LIN {X 226.458,Y -181.154,Z 168.975,A 141.342,B 90.000,C 0.000} C_DIS
LIN {X 226.330,Y -181.313,Z 169.018,A 141.302,B 90.000,C 0.000} C_DIS
LIN {X 226.304,Y -181.347,Z 169.069,A 141.293,B 90.000,C 0.000} C_DIS
LIN {X 226.264,Y -181.396,Z 169.120,A 141.281,B 90.000,C 0.000} C_DIS
LIN {X 226.072,Y -181.635,Z 169.162,A 141.220,B 90.000,C 0.000} C_DIS
LIN {X 225.993,Y -181.734,Z 169.264,A 141.195,B 90.000,C 0.000} C_DIS
LIN {X 225.801,Y -181.973,Z 169.307,A 141.135,B 90.000,C 0.000} C_DIS
LIN {X 225.721,Y -182.072,Z 169.409,A 141.109,B 90.000,C 0.000} C_DIS
LIN {X 225.528,Y -182.310,Z 169.451,A 141.049,B 90.000,C 0.000} C_DIS
LIN {X 225.488,Y -182.360,Z 169.502,A 141.036,B 90.000,C 0.000} C_DIS
LIN {X 225.461,Y -182.393,Z 169.554,A 141.028,B 90.000,C 0.000} C_DIS
LIN {X 225.333,Y -182.551,Z 169.596,A 140.988,B 90.000,C 0.000} C_DIS
LIN {X 225.306,Y -182.584,Z 169.647,A 140.979,B 90.000,C 0.000} C_DIS
LIN {X 225.266,Y -182.634,Z 169.698,A 140.967,B 90.000,C 0.000} C_DIS
LIN {X 225.073,Y -182.872,Z 169.740,A 140.906,B 90.000,C 0.000} C_DIS
LIN {X 224.993,Y -182.970,Z 169.843,A 140.881,B 90.000,C 0.000} C_DIS
LIN {X 224.800,Y -183.208,Z 169.885,A 140.821,B 90.000,C 0.000} C_DIS
LIN {X 224.719,Y -183.307,Z 169.987,A 140.795,B 90.000,C 0.000} C_DIS
LIN {X 224.525,Y -183.544,Z 170.030,A 140.735,B 90.000,C 0.000} C_DIS
LIN {X 224.445,Y -183.642,Z 170.132,A 140.710,B 90.000,C 0.000} C_DIS
LIN {X 224.251,Y -183.879,Z 170.174,A 140.649,B 90.000,C 0.000} C_DIS
LIN {X 224.210,Y -183.929,Z 170.225,A 140.637,B 90.000,C 0.000} C_DIS
LIN {X 224.183,Y -183.961,Z 170.276,A 140.628,B 90.000,C 0.000} C_DIS
LIN {X 224.054,Y -184.119,Z 170.319,A 140.588,B 90.000,C 0.000} C_DIS
LIN {X 224.027,Y -184.152,Z 170.370,A 140.580,B 90.000,C 0.000} C_DIS
LIN {X 223.986,Y -184.201,Z 170.421,A 140.567,B 90.000,C 0.000} C_DIS
LIN {X 223.792,Y -184.438,Z 170.463,A 140.506,B 90.000,C 0.000} C_DIS
LIN {X 223.711,Y -184.536,Z 170.565,A 140.481,B 90.000,C 0.000} C_DIS
LIN {X 223.516,Y -184.772,Z 170.608,A 140.421,B 90.000,C 0.000} C_DIS
LIN {X 223.435,Y -184.870,Z 170.710,A 140.396,B 90.000,C 0.000} C_DIS
LIN {X 223.239,Y -185.106,Z 170.752,A 140.335,B 90.000,C 0.000} C_DIS
LIN {X 223.199,Y -185.155,Z 170.803,A 140.323,B 90.000,C 0.000} C_DIS
LIN {X 223.172,Y -185.188,Z 170.854,A 140.314,B 90.000,C 0.000} C_DIS
LIN {X 223.041,Y -185.345,Z 170.897,A 140.274,B 90.000,C 0.000} C_DIS
LIN {X 223.014,Y -185.377,Z 170.948,A 140.265,B 90.000,C 0.000} C_DIS
LIN {X 222.973,Y -185.426,Z 170.999,A 140.253,B 90.000,C 0.000} C_DIS
LIN {X 222.777,Y -185.662,Z 171.041,A 140.192,B 90.000,C 0.000} C_DIS
LIN {X 222.696,Y -185.759,Z 171.143,A 140.167,B 90.000,C 0.000} C_DIS
LIN {X 222.500,Y -185.995,Z 171.186,A 140.107,B 90.000,C 0.000} C_DIS
LIN {X 222.418,Y -186.092,Z 171.288,A 140.082,B 90.000,C 0.000} C_DIS
LIN {X 222.221,Y -186.327,Z 171.330,A 140.021,B 90.000,C 0.000} C_DIS
LIN {X 222.180,Y -186.376,Z 171.381,A 140.008,B 90.000,C 0.000} C_DIS
LIN {X 222.153,Y -186.408,Z 171.432,A 140.000,B 90.000,C 0.000} C_DIS
LIN {X 222.022,Y -186.565,Z 171.475,A 139.960,B 90.000,C 0.000} C_DIS
LIN {X 221.994,Y -186.597,Z 171.526,A 139.951,B 90.000,C 0.000} C_DIS
LIN {X 221.953,Y -186.646,Z 171.577,A 139.939,B 90.000,C 0.000} C_DIS
LIN {X 221.756,Y -186.880,Z 171.619,A 139.878,B 90.000,C 0.000} C_DIS
LIN {X 221.674,Y -186.977,Z 171.721,A 139.853,B 90.000,C 0.000} C_DIS
LIN {X 221.477,Y -187.211,Z 171.764,A 139.793,B 90.000,C 0.000} C_DIS
LIN {X 221.394,Y -187.309,Z 171.866,A 139.767,B 90.000,C 0.000} C_DIS
LIN {X 221.196,Y -187.542,Z 171.908,A 139.707,B 90.000,C 0.000} C_DIS
LIN {X 221.114,Y -187.640,Z 172.010,A 139.682,B 90.000,C 0.000} C_DIS
LIN {X 220.916,Y -187.873,Z 172.053,A 139.621,B 90.000,C 0.000} C_DIS
LIN {X 220.875,Y -187.921,Z 172.104,A 139.609,B 90.000,C 0.000} C_DIS
LIN {X 220.847,Y -187.954,Z 172.155,A 139.600,B 90.000,C 0.000} C_DIS
LIN {X 220.715,Y -188.109,Z 172.197,A 139.560,B 90.000,C 0.000} C_DIS
LIN {X 220.687,Y -188.141,Z 172.249,A 139.552,B 90.000,C 0.000} C_DIS
LIN {X 220.646,Y -188.190,Z 172.300,A 139.539,B 90.000,C 0.000} C_DIS
LIN {X 220.447,Y -188.423,Z 172.342,A 139.478,B 90.000,C 0.000} C_DIS
LIN {X 220.364,Y -188.520,Z 172.444,A 139.453,B 90.000,C 0.000} C_DIS
LIN {X 220.165,Y -188.752,Z 172.487,A 139.393,B 90.000,C 0.000} C_DIS
LIN {X 220.082,Y -188.849,Z 172.589,A 139.368,B 90.000,C 0.000} C_DIS
LIN {X 219.883,Y -189.081,Z 172.631,A 139.307,B 90.000,C 0.000} C_DIS
LIN {X 219.841,Y -189.129,Z 172.682,A 139.295,B 90.000,C 0.000} C_DIS
LIN {X 219.813,Y -189.162,Z 172.733,A 139.286,B 90.000,C 0.000} C_DIS
LIN {X 219.680,Y -189.316,Z 172.776,A 139.246,B 90.000,C 0.000} C_DIS
LIN {X 219.652,Y -189.348,Z 172.827,A 139.237,B 90.000,C 0.000} C_DIS
LIN {X 219.611,Y -189.397,Z 172.878,A 139.225,B 90.000,C 0.000} C_DIS
LIN {X 219.411,Y -189.628,Z 172.920,A 139.164,B 90.000,C 0.000} C_DIS
LIN {X 219.327,Y -189.725,Z 173.022,A 139.139,B 90.000,C 0.000} C_DIS
LIN {X 219.127,Y -189.956,Z 173.065,A 139.079,B 90.000,C 0.000} C_DIS
LIN {X 219.043,Y -190.053,Z 173.167,A 139.054,B 90.000,C 0.000} C_DIS
LIN {X 218.843,Y -190.284,Z 173.209,A 138.993,B 90.000,C 0.000} C_DIS
LIN {X 218.801,Y -190.332,Z 173.260,A 138.980,B 90.000,C 0.000} C_DIS
LIN {X 218.773,Y -190.364,Z 173.311,A 138.972,B 90.000,C 0.000} C_DIS
LIN {X 218.639,Y -190.518,Z 173.354,A 138.932,B 90.000,C 0.000} C_DIS
LIN {X 218.611,Y -190.550,Z 173.405,A 138.923,B 90.000,C 0.000} C_DIS
LIN {X 218.569,Y -190.598,Z 173.456,A 138.911,B 90.000,C 0.000} C_DIS
LIN {X 218.368,Y -190.828,Z 173.498,A 138.850,B 90.000,C 0.000} C_DIS
LIN {X 218.284,Y -190.924,Z 173.600,A 138.825,B 90.000,C 0.000} C_DIS
LIN {X 218.082,Y -191.155,Z 173.643,A 138.765,B 90.000,C 0.000} C_DIS
LIN {X 217.998,Y -191.250,Z 173.745,A 138.739,B 90.000,C 0.000} C_DIS
LIN {X 217.796,Y -191.481,Z 173.787,A 138.679,B 90.000,C 0.000} C_DIS
LIN {X 217.712,Y -191.576,Z 173.889,A 138.654,B 90.000,C 0.000} C_DIS
LIN {X 217.510,Y -191.806,Z 173.932,A 138.593,B 90.000,C 0.000} C_DIS
LIN {X 217.468,Y -191.854,Z 173.983,A 138.581,B 90.000,C 0.000} C_DIS
LIN {X 217.439,Y -191.886,Z 174.034,A 138.572,B 90.000,C 0.000} C_DIS
LIN {X 217.304,Y -192.039,Z 174.076,A 138.532,B 90.000,C 0.000} C_DIS
LIN {X 217.276,Y -192.070,Z 174.127,A 138.524,B 90.000,C 0.000} C_DIS
LIN {X 217.234,Y -192.118,Z 174.178,A 138.511,B 90.000,C 0.000} C_DIS
LIN {X 217.031,Y -192.347,Z 174.221,A 138.450,B 90.000,C 0.000} C_DIS
LIN {X 216.947,Y -192.443,Z 174.323,A 138.425,B 90.000,C 0.000} C_DIS
LIN {X 216.743,Y -192.672,Z 174.365,A 138.365,B 90.000,C 0.000} C_DIS
LIN {X 216.659,Y -192.767,Z 174.467,A 138.340,B 90.000,C 0.000} C_DIS
LIN {X 216.455,Y -192.996,Z 174.510,A 138.279,B 90.000,C 0.000} C_DIS
LIN {X 216.413,Y -193.043,Z 174.561,A 138.267,B 90.000,C 0.000} C_DIS
LIN {X 216.384,Y -193.075,Z 174.612,A 138.258,B 90.000,C 0.000} C_DIS
LIN {X 216.248,Y -193.227,Z 174.654,A 138.218,B 90.000,C 0.000} C_DIS
LIN {X 216.220,Y -193.259,Z 174.705,A 138.209,B 90.000,C 0.000} C_DIS
LIN {X 216.178,Y -193.306,Z 174.757,A 138.197,B 90.000,C 0.000} C_DIS
LIN {X 215.973,Y -193.534,Z 174.799,A 138.136,B 90.000,C 0.000} C_DIS
LIN {X 215.888,Y -193.629,Z 174.901,A 138.111,B 90.000,C 0.000} C_DIS
LIN {X 215.684,Y -193.857,Z 174.944,A 138.051,B 90.000,C 0.000} C_DIS
LIN {X 215.599,Y -193.952,Z 175.046,A 138.026,B 90.000,C 0.000} C_DIS
LIN {X 215.394,Y -194.179,Z 175.088,A 137.965,B 90.000,C 0.000} C_DIS
LIN {X 215.351,Y -194.227,Z 175.139,A 137.952,B 90.000,C 0.000} C_DIS
LIN {X 215.323,Y -194.258,Z 175.190,A 137.944,B 90.000,C 0.000} C_DIS
LIN {X 215.186,Y -194.410,Z 175.233,A 137.904,B 90.000,C 0.000} C_DIS
LIN {X 215.157,Y -194.441,Z 175.284,A 137.895,B 90.000,C 0.000} C_DIS
LIN {X 215.115,Y -194.488,Z 175.335,A 137.883,B 90.000,C 0.000} C_DIS
LIN {X 214.909,Y -194.715,Z 175.377,A 137.822,B 90.000,C 0.000} C_DIS
LIN {X 214.824,Y -194.810,Z 175.479,A 137.797,B 90.000,C 0.000} C_DIS
LIN {X 214.618,Y -195.036,Z 175.522,A 137.737,B 90.000,C 0.000} C_DIS
LIN {X 214.532,Y -195.131,Z 175.624,A 137.711,B 90.000,C 0.000} C_DIS
LIN {X 214.326,Y -195.357,Z 175.666,A 137.651,B 90.000,C 0.000} C_DIS
LIN {X 214.283,Y -195.404,Z 175.717,A 137.638,B 90.000,C 0.000} C_DIS
LIN {X 214.254,Y -195.436,Z 175.768,A 137.630,B 90.000,C 0.000} C_DIS
LIN {X 214.117,Y -195.586,Z 175.811,A 137.590,B 90.000,C 0.000} C_DIS
LIN {X 214.088,Y -195.618,Z 175.862,A 137.581,B 90.000,C 0.000} C_DIS
LIN {X 214.045,Y -195.665,Z 175.913,A 137.569,B 90.000,C 0.000} C_DIS
LIN {X 213.838,Y -195.891,Z 175.955,A 137.508,B 90.000,C 0.000} C_DIS
LIN {X 213.752,Y -195.984,Z 176.057,A 137.483,B 90.000,C 0.000} C_DIS
LIN {X 213.545,Y -196.210,Z 176.100,A 137.423,B 90.000,C 0.000} C_DIS
LIN {X 213.459,Y -196.304,Z 176.202,A 137.397,B 90.000,C 0.000} C_DIS
LIN {X 213.252,Y -196.529,Z 176.244,A 137.337,B 90.000,C 0.000} C_DIS
LIN {X 213.209,Y -196.576,Z 176.295,A 137.324,B 90.000,C 0.000} C_DIS
LIN {X 213.180,Y -196.607,Z 176.346,A 137.316,B 90.000,C 0.000} C_DIS
LIN {X 213.041,Y -196.757,Z 176.389,A 137.276,B 90.000,C 0.000} C_DIS
LIN {X 213.013,Y -196.788,Z 176.440,A 137.267,B 90.000,C 0.000} C_DIS
LIN {X 212.969,Y -196.835,Z 176.491,A 137.255,B 90.000,C 0.000} C_DIS
LIN {X 212.761,Y -197.060,Z 176.533,A 137.194,B 90.000,C 0.000} C_DIS
LIN {X 212.675,Y -197.153,Z 176.635,A 137.169,B 90.000,C 0.000} C_DIS
LIN {X 212.466,Y -197.378,Z 176.678,A 137.108,B 90.000,C 0.000} C_DIS
LIN {X 212.380,Y -197.471,Z 176.780,A 137.083,B 90.000,C 0.000} C_DIS
LIN {X 212.171,Y -197.695,Z 176.822,A 137.023,B 90.000,C 0.000} C_DIS
LIN {X 212.084,Y -197.788,Z 176.924,A 136.998,B 90.000,C 0.000} C_DIS
LIN {X 211.875,Y -198.012,Z 176.967,A 136.937,B 90.000,C 0.000} C_DIS
LIN {X 211.832,Y -198.059,Z 177.018,A 136.925,B 90.000,C 0.000} C_DIS
LIN {X 211.803,Y -198.090,Z 177.069,A 136.916,B 90.000,C 0.000} C_DIS
LIN {X 211.663,Y -198.239,Z 177.111,A 136.876,B 90.000,C 0.000} C_DIS
LIN {X 211.634,Y -198.270,Z 177.162,A 136.867,B 90.000,C 0.000} C_DIS
LIN {X 211.591,Y -198.316,Z 177.213,A 136.855,B 90.000,C 0.000} C_DIS
LIN {X 211.381,Y -198.540,Z 177.256,A 136.794,B 90.000,C 0.000} C_DIS
LIN {X 211.294,Y -198.632,Z 177.358,A 136.769,B 90.000,C 0.000} C_DIS
LIN {X 211.084,Y -198.855,Z 177.400,A 136.709,B 90.000,C 0.000} C_DIS
LIN {X 210.997,Y -198.948,Z 177.503,A 136.683,B 90.000,C 0.000} C_DIS
LIN {X 210.787,Y -199.171,Z 177.545,A 136.623,B 90.000,C 0.000} C_DIS
LIN {X 210.743,Y -199.217,Z 177.596,A 136.610,B 90.000,C 0.000} C_DIS
LIN {X 210.714,Y -199.248,Z 177.647,A 136.602,B 90.000,C 0.000} C_DIS
LIN {X 210.573,Y -199.396,Z 177.690,A 136.562,B 90.000,C 0.000} C_DIS
LIN {X 210.544,Y -199.427,Z 177.741,A 136.553,B 90.000,C 0.000} C_DIS
LIN {X 210.500,Y -199.473,Z 177.792,A 136.541,B 90.000,C 0.000} C_DIS
LIN {X 210.290,Y -199.695,Z 177.834,A 136.480,B 90.000,C 0.000} C_DIS
LIN {X 210.202,Y -199.788,Z 177.936,A 136.455,B 90.000,C 0.000} C_DIS
LIN {X 209.991,Y -200.010,Z 177.979,A 136.395,B 90.000,C 0.000} C_DIS
LIN {X 209.903,Y -200.102,Z 178.081,A 136.369,B 90.000,C 0.000} C_DIS
LIN {X 209.692,Y -200.323,Z 178.123,A 136.309,B 90.000,C 0.000} C_DIS
LIN {X 209.604,Y -200.415,Z 178.225,A 136.284,B 90.000,C 0.000} C_DIS
LIN {X 209.392,Y -200.637,Z 178.268,A 136.223,B 90.000,C 0.000} C_DIS
LIN {X 209.348,Y -200.683,Z 178.319,A 136.211,B 90.000,C 0.000} C_DIS
LIN {X 209.318,Y -200.713,Z 178.370,A 136.202,B 90.000,C 0.000} C_DIS
LIN {X 209.177,Y -200.861,Z 178.412,A 136.162,B 90.000,C 0.000} C_DIS
LIN {X 209.148,Y -200.891,Z 178.463,A 136.154,B 90.000,C 0.000} C_DIS
LIN {X 209.104,Y -200.937,Z 178.514,A 136.141,B 90.000,C 0.000} C_DIS
LIN {X 208.891,Y -201.158,Z 178.557,A 136.080,B 90.000,C 0.000} C_DIS
LIN {X 208.803,Y -201.250,Z 178.659,A 136.055,B 90.000,C 0.000} C_DIS
LIN {X 208.590,Y -201.470,Z 178.701,A 135.995,B 90.000,C 0.000} C_DIS
LIN {X 208.502,Y -201.561,Z 178.803,A 135.970,B 90.000,C 0.000} C_DIS
LIN {X 208.289,Y -201.782,Z 178.846,A 135.909,B 90.000,C 0.000} C_DIS
LIN {X 208.244,Y -201.827,Z 178.897,A 135.897,B 90.000,C 0.000} C_DIS
LIN {X 208.215,Y -201.858,Z 178.948,A 135.888,B 90.000,C 0.000} C_DIS
LIN {X 208.073,Y -202.004,Z 178.990,A 135.848,B 90.000,C 0.000} C_DIS
LIN {X 208.043,Y -202.035,Z 179.041,A 135.839,B 90.000,C 0.000} C_DIS
LIN {X 207.999,Y -202.080,Z 179.092,A 135.827,B 90.000,C 0.000} C_DIS
LIN {X 207.790,Y -202.295,Z 179.127,A 135.768,B 90.000,C 0.000} C_DIS
LIN {X 207.748,Y -202.338,Z 179.167,A 135.756,B 90.000,C 0.000} C_DIS
LIN {X 207.765,Y -202.321,Z 179.235,A 135.761,B 90.000,C 0.000} C_DIS
LIN {X 207.913,Y -202.169,Z 179.437,A 135.802,B 90.000,C 0.000} C_DIS
LIN {X 207.972,Y -202.108,Z 179.657,A 135.819,B 90.000,C 0.000} C_DIS
LIN {X 208.114,Y -201.961,Z 179.875,A 135.860,B 90.000,C 0.000} C_DIS
LIN {X 208.144,Y -201.931,Z 179.997,A 135.868,B 90.000,C 0.000} C_DIS
LIN {X 208.159,Y -201.916,Z 180.088,A 135.872,B 90.000,C 0.000} C_DIS
LIN {X 208.230,Y -201.842,Z 180.168,A 135.892,B 90.000,C 0.000} C_DIS
LIN {X 208.259,Y -201.812,Z 180.372,A 135.901,B 90.000,C 0.000} C_DIS
LIN {X 208.330,Y -201.739,Z 180.457,A 135.921,B 90.000,C 0.000} C_DIS
LIN {X 208.360,Y -201.708,Z 180.661,A 135.929,B 90.000,C 0.000} C_DIS
LIN {X 208.431,Y -201.635,Z 180.746,A 135.949,B 90.000,C 0.000} C_DIS
LIN {X 208.460,Y -201.604,Z 180.950,A 135.958,B 90.000,C 0.000} C_DIS
LIN {X 208.496,Y -201.568,Z 180.992,A 135.968,B 90.000,C 0.000} C_DIS
LIN {X 208.531,Y -201.531,Z 181.056,A 135.978,B 90.000,C 0.000} C_DIS
LIN {X 208.561,Y -201.500,Z 181.362,A 135.986,B 90.000,C 0.000} C_DIS
LIN {X 208.596,Y -201.464,Z 181.426,A 135.996,B 90.000,C 0.000} C_DIS
LIN {X 208.632,Y -201.427,Z 181.511,A 136.007,B 90.000,C 0.000} C_DIS
LIN {X 208.661,Y -201.396,Z 181.919,A 136.015,B 90.000,C 0.000} C_DIS
LIN {X 208.697,Y -201.360,Z 182.004,A 136.025,B 90.000,C 0.000} C_DIS
LIN {X 208.733,Y -201.321,Z 182.329,A 136.036,B 90.000,C 0.000} C_DIS
LIN {X 208.733,Y -201.321,Z 184.136,A 136.036,B 90.000,C 0.000} C_DIS
LIN {X 208.697,Y -201.360,Z 184.461,A 136.025,B 90.000,C 0.000} C_DIS
LIN {X 208.661,Y -201.396,Z 184.546,A 136.015,B 90.000,C 0.000} C_DIS
LIN {X 208.632,Y -201.427,Z 184.954,A 136.007,B 90.000,C 0.000} C_DIS
LIN {X 208.596,Y -201.464,Z 185.039,A 135.996,B 90.000,C 0.000} C_DIS
LIN {X 208.561,Y -201.500,Z 185.103,A 135.986,B 90.000,C 0.000} C_DIS
LIN {X 208.531,Y -201.531,Z 185.409,A 135.978,B 90.000,C 0.000} C_DIS
LIN {X 208.496,Y -201.568,Z 185.473,A 135.968,B 90.000,C 0.000} C_DIS
LIN {X 208.460,Y -201.604,Z 185.515,A 135.958,B 90.000,C 0.000} C_DIS
LIN {X 208.431,Y -201.635,Z 185.719,A 135.949,B 90.000,C 0.000} C_DIS
LIN {X 208.360,Y -201.708,Z 185.804,A 135.929,B 90.000,C 0.000} C_DIS
LIN {X 208.330,Y -201.739,Z 186.008,A 135.921,B 90.000,C 0.000} C_DIS
LIN {X 208.259,Y -201.812,Z 186.093,A 135.901,B 90.000,C 0.000} C_DIS
LIN {X 208.230,Y -201.842,Z 186.298,A 135.892,B 90.000,C 0.000} C_DIS
LIN {X 208.194,Y -201.879,Z 186.340,A 135.882,B 90.000,C 0.000} C_DIS
LIN {X 208.159,Y -201.916,Z 186.374,A 135.872,B 90.000,C 0.000} C_DIS
LIN {X 208.144,Y -201.931,Z 186.456,A 135.868,B 90.000,C 0.000} C_DIS
LIN {X 208.100,Y -201.977,Z 186.597,A 135.855,B 90.000,C 0.000} C_DIS
LIN {X 207.741,Y -202.346,Z 187.263,A 135.754,B 90.000,C 0.000} C_DIS
LIN {X 207.268,Y -202.830,Z 187.931,A 135.620,B 90.000,C 0.000} C_DIS
LIN {X 206.983,Y -203.121,Z 188.219,A 135.540,B 90.000,C 0.000} C_DIS
LIN {X 206.908,Y -203.197,Z 188.321,A 135.519,B 90.000,C 0.000} C_DIS
LIN {X 206.754,Y -203.354,Z 188.406,A 135.475,B 90.000,C 0.000} C_DIS
LIN {X 206.601,Y -203.509,Z 188.610,A 135.432,B 90.000,C 0.000} C_DIS
LIN {X 206.516,Y -203.596,Z 188.652,A 135.408,B 90.000,C 0.000} C_DIS
LIN {X 206.452,Y -203.660,Z 188.674,A 135.390,B 90.000,C 0.000} C_DIS
LIN {X 206.396,Y -203.717,Z 188.776,A 135.374,B 90.000,C 0.000} C_DIS
LIN {X 206.252,Y -203.863,Z 188.818,A 135.334,B 90.000,C 0.000} C_DIS
LIN {X 206.222,Y -203.893,Z 188.869,A 135.325,B 90.000,C 0.000} C_DIS
LIN {X 206.178,Y -203.938,Z 188.920,A 135.313,B 90.000,C 0.000} C_DIS
LIN {X 205.962,Y -204.156,Z 188.963,A 135.252,B 90.000,C 0.000} C_DIS
LIN {X 205.873,Y -204.246,Z 189.065,A 135.227,B 90.000,C 0.000} C_DIS
LIN {X 205.657,Y -204.463,Z 189.107,A 135.167,B 90.000,C 0.000} C_DIS
LIN {X 205.612,Y -204.509,Z 189.158,A 135.154,B 90.000,C 0.000} C_DIS
LIN {X 205.552,Y -204.569,Z 189.209,A 135.137,B 90.000,C 0.000} C_DIS
LIN {X 205.264,Y -204.858,Z 189.252,A 135.057,B 90.000,C 0.000} C_DIS
LIN {X 205.204,Y -204.918,Z 189.303,A 135.040,B 90.000,C 0.000} C_DIS
LIN {X 204.999,Y -205.123,Z 189.356,A 134.983,B 90.000,C 0.000} C_DIS
LIN {X 203.872,Y -206.243,Z 189.356,A 134.669,B 90.000,C 0.000} C_DIS
LIN {X 203.666,Y -206.446,Z 189.303,A 134.612,B 90.000,C 0.000} C_DIS
LIN {X 203.591,Y -206.521,Z 189.252,A 134.591,B 90.000,C 0.000} C_DIS
LIN {X 203.227,Y -206.879,Z 189.209,A 134.490,B 90.000,C 0.000} C_DIS
LIN {X 203.151,Y -206.953,Z 189.158,A 134.469,B 90.000,C 0.000} C_DIS
LIN {X 203.106,Y -206.998,Z 189.107,A 134.456,B 90.000,C 0.000} C_DIS
LIN {X 202.887,Y -207.212,Z 189.065,A 134.396,B 90.000,C 0.000} C_DIS
LIN {X 202.841,Y -207.257,Z 189.014,A 134.383,B 90.000,C 0.000} C_DIS
LIN {X 202.811,Y -207.286,Z 188.963,A 134.375,B 90.000,C 0.000} C_DIS
LIN {X 202.665,Y -207.429,Z 188.920,A 134.334,B 90.000,C 0.000} C_DIS
LIN {X 202.604,Y -207.488,Z 188.818,A 134.318,B 90.000,C 0.000} C_DIS
LIN {X 202.458,Y -207.631,Z 188.776,A 134.277,B 90.000,C 0.000} C_DIS
LIN {X 202.397,Y -207.690,Z 188.674,A 134.261,B 90.000,C 0.000} C_DIS
LIN {X 202.251,Y -207.833,Z 188.631,A 134.220,B 90.000,C 0.000} C_DIS
LIN {X 202.221,Y -207.862,Z 188.580,A 134.212,B 90.000,C 0.000} C_DIS
LIN {X 202.196,Y -207.886,Z 188.529,A 134.205,B 90.000,C 0.000} C_DIS
LIN {X 202.138,Y -207.943,Z 188.508,A 134.189,B 90.000,C 0.000} C_DIS
LIN {X 202.037,Y -208.041,Z 188.444,A 134.161,B 90.000,C 0.000} C_DIS
LIN {X 201.259,Y -208.794,Z 187.569,A 133.947,B 90.000,C 0.000} C_DIS
LIN {X 201.108,Y -208.939,Z 187.496,A 133.906,B 90.000,C 0.000} C_DIS
LIN {X 201.014,Y -209.030,Z 187.517,A 133.880,B 90.000,C 0.000} C_DIS
LIN {X 200.974,Y -209.068,Z 187.568,A 133.869,B 90.000,C 0.000} C_DIS
LIN {X 200.913,Y -209.127,Z 187.620,A 133.852,B 90.000,C 0.000} C_DIS
LIN {X 200.618,Y -209.410,Z 187.662,A 133.772,B 90.000,C 0.000} C_DIS
LIN {X 200.557,Y -209.468,Z 187.713,A 133.755,B 90.000,C 0.000} C_DIS
LIN {X 200.511,Y -209.512,Z 187.764,A 133.742,B 90.000,C 0.000} C_DIS
LIN {X 200.290,Y -209.724,Z 187.807,A 133.682,B 90.000,C 0.000} C_DIS
LIN {X 200.243,Y -209.768,Z 187.858,A 133.669,B 90.000,C 0.000} C_DIS
LIN {X 200.182,Y -209.826,Z 187.909,A 133.653,B 90.000,C 0.000} C_DIS
LIN {X 199.886,Y -210.108,Z 187.951,A 133.572,B 90.000,C 0.000} C_DIS
LIN {X 199.825,Y -210.167,Z 188.002,A 133.555,B 90.000,C 0.000} C_DIS
LIN {X 199.779,Y -210.210,Z 188.053,A 133.542,B 90.000,C 0.000} C_DIS
LIN {X 199.557,Y -210.421,Z 188.096,A 133.482,B 90.000,C 0.000} C_DIS
LIN {X 199.510,Y -210.465,Z 188.147,A 133.469,B 90.000,C 0.000} C_DIS
LIN {X 199.449,Y -210.524,Z 188.198,A 133.453,B 90.000,C 0.000} C_DIS
LIN {X 199.152,Y -210.804,Z 188.240,A 133.372,B 90.000,C 0.000} C_DIS
LIN {X 199.090,Y -210.862,Z 188.291,A 133.355,B 90.000,C 0.000} C_DIS
LIN {X 199.044,Y -210.906,Z 188.342,A 133.343,B 90.000,C 0.000} C_DIS
LIN {X 198.821,Y -211.116,Z 188.385,A 133.282,B 90.000,C 0.000} C_DIS
LIN {X 198.729,Y -211.204,Z 188.487,A 133.257,B 90.000,C 0.000} C_DIS
LIN {X 198.506,Y -211.413,Z 188.529,A 133.196,B 90.000,C 0.000} C_DIS
LIN {X 198.459,Y -211.457,Z 188.580,A 133.184,B 90.000,C 0.000} C_DIS
LIN {X 198.367,Y -211.543,Z 188.631,A 133.159,B 90.000,C 0.000} C_DIS
LIN {X 197.918,Y -211.963,Z 188.674,A 133.038,B 90.000,C 0.000} C_DIS
LIN {X 197.826,Y -212.049,Z 188.725,A 133.013,B 90.000,C 0.000} C_DIS
LIN {X 197.795,Y -212.078,Z 188.776,A 133.004,B 90.000,C 0.000} C_DIS
LIN {X 197.720,Y -212.148,Z 188.797,A 132.984,B 90.000,C 0.000} C_DIS
LIN {X 197.645,Y -212.217,Z 188.776,A 132.964,B 90.000,C 0.000} C_DIS
LIN {X 197.614,Y -212.246,Z 188.725,A 132.955,B 90.000,C 0.000} C_DIS
LIN {X 197.537,Y -212.319,Z 188.674,A 132.934,B 90.000,C 0.000} C_DIS
LIN {X 197.163,Y -212.666,Z 188.631,A 132.834,B 90.000,C 0.000} C_DIS
LIN {X 197.085,Y -212.738,Z 188.580,A 132.813,B 90.000,C 0.000} C_DIS
LIN {X 197.061,Y -212.760,Z 188.529,A 132.806,B 90.000,C 0.000} C_DIS
LIN {X 197.004,Y -212.813,Z 188.508,A 132.791,B 90.000,C 0.000} C_DIS
LIN {X 196.873,Y -212.935,Z 188.410,A 132.756,B 90.000,C 0.000} C_DIS
LIN {X 196.687,Y -213.106,Z 188.183,A 132.705,B 90.000,C 0.000} C_DIS
LIN {X 196.520,Y -213.260,Z 187.930,A 132.661,B 90.000,C 0.000} C_DIS
LIN {X 196.448,Y -213.327,Z 187.751,A 132.641,B 90.000,C 0.000} C_DIS
LIN {X 196.432,Y -213.341,Z 187.673,A 132.637,B 90.000,C 0.000} C_DIS
LIN {X 196.395,Y -213.376,Z 187.641,A 132.627,B 90.000,C 0.000} C_DIS
LIN {X 196.356,Y -213.411,Z 187.460,A 132.617,B 90.000,C 0.000} C_DIS
LIN {X 196.356,Y -213.411,Z 186.521,A 132.617,B 90.000,C 0.000} C_DIS
LIN {X 196.395,Y -213.376,Z 186.340,A 132.627,B 90.000,C 0.000} C_DIS
LIN {X 196.432,Y -213.341,Z 186.298,A 132.637,B 90.000,C 0.000} C_DIS
LIN {X 196.464,Y -213.312,Z 186.093,A 132.646,B 90.000,C 0.000} C_DIS
LIN {X 196.501,Y -213.278,Z 186.051,A 132.656,B 90.000,C 0.000} C_DIS
LIN {X 196.539,Y -213.243,Z 186.019,A 132.666,B 90.000,C 0.000} C_DIS
LIN {X 196.554,Y -213.229,Z 185.941,A 132.670,B 90.000,C 0.000} C_DIS
LIN {X 196.626,Y -213.163,Z 185.766,A 132.689,B 90.000,C 0.000} C_DIS
LIN {X 196.973,Y -212.842,Z 185.283,A 132.782,B 90.000,C 0.000} C_DIS
LIN {X 197.244,Y -212.591,Z 185.039,A 132.855,B 90.000,C 0.000} C_DIS
LIN {X 197.326,Y -212.515,Z 184.937,A 132.877,B 90.000,C 0.000} C_DIS
LIN {X 197.414,Y -212.432,Z 184.895,A 132.901,B 90.000,C 0.000} C_DIS
LIN {X 197.481,Y -212.371,Z 184.873,A 132.919,B 90.000,C 0.000} C_DIS
LIN {X 197.540,Y -212.316,Z 184.771,A 132.935,B 90.000,C 0.000} C_DIS
LIN {X 197.689,Y -212.177,Z 184.729,A 132.976,B 90.000,C 0.000} C_DIS
LIN {X 197.751,Y -212.119,Z 184.627,A 132.992,B 90.000,C 0.000} C_DIS
LIN {X 197.901,Y -211.980,Z 184.584,A 133.033,B 90.000,C 0.000} C_DIS
LIN {X 197.963,Y -211.922,Z 184.482,A 133.049,B 90.000,C 0.000} C_DIS
LIN {X 198.112,Y -211.782,Z 184.440,A 133.090,B 90.000,C 0.000} C_DIS
LIN {X 198.174,Y -211.724,Z 184.338,A 133.107,B 90.000,C 0.000} C_DIS
LIN {X 198.323,Y -211.585,Z 184.295,A 133.147,B 90.000,C 0.000} C_DIS
LIN {X 198.354,Y -211.556,Z 184.244,A 133.155,B 90.000,C 0.000} C_DIS
LIN {X 198.400,Y -211.512,Z 184.193,A 133.168,B 90.000,C 0.000} C_DIS
LIN {X 198.623,Y -211.303,Z 184.151,A 133.228,B 90.000,C 0.000} C_DIS
LIN {X 198.670,Y -211.259,Z 184.100,A 133.241,B 90.000,C 0.000} C_DIS
LIN {X 198.701,Y -211.230,Z 184.049,A 133.249,B 90.000,C 0.000} C_DIS
LIN {X 198.849,Y -211.090,Z 184.006,A 133.290,B 90.000,C 0.000} C_DIS
LIN {X 198.911,Y -211.032,Z 183.904,A 133.306,B 90.000,C 0.000} C_DIS
LIN {X 199.060,Y -210.892,Z 183.862,A 133.347,B 90.000,C 0.000} C_DIS
LIN {X 199.121,Y -210.833,Z 183.760,A 133.364,B 90.000,C 0.000} C_DIS
LIN {X 199.270,Y -210.693,Z 183.717,A 133.404,B 90.000,C 0.000} C_DIS
LIN {X 199.331,Y -210.635,Z 183.615,A 133.421,B 90.000,C 0.000} C_DIS
LIN {X 199.480,Y -210.494,Z 183.573,A 133.461,B 90.000,C 0.000} C_DIS
LIN {X 199.541,Y -210.436,Z 183.471,A 133.478,B 90.000,C 0.000} C_DIS
LIN {X 199.689,Y -210.295,Z 183.428,A 133.518,B 90.000,C 0.000} C_DIS
LIN {X 199.751,Y -210.237,Z 183.326,A 133.535,B 90.000,C 0.000} C_DIS
LIN {X 199.899,Y -210.096,Z 183.284,A 133.575,B 90.000,C 0.000} C_DIS
LIN {X 199.930,Y -210.067,Z 183.233,A 133.584,B 90.000,C 0.000} C_DIS
LIN {X 199.899,Y -210.096,Z 183.182,A 133.575,B 90.000,C 0.000} C_DIS
LIN {X 199.825,Y -210.167,Z 183.160,A 133.555,B 90.000,C 0.000} C_DIS
LIN {X 199.751,Y -210.237,Z 183.182,A 133.535,B 90.000,C 0.000} C_DIS
LIN {X 199.689,Y -210.295,Z 183.284,A 133.518,B 90.000,C 0.000} C_DIS
LIN {X 199.541,Y -210.436,Z 183.326,A 133.478,B 90.000,C 0.000} C_DIS
LIN {X 199.510,Y -210.465,Z 183.377,A 133.469,B 90.000,C 0.000} C_DIS
LIN {X 199.464,Y -210.509,Z 183.428,A 133.457,B 90.000,C 0.000} C_DIS
LIN {X 199.242,Y -210.719,Z 183.471,A 133.396,B 90.000,C 0.000} C_DIS
LIN {X 199.149,Y -210.807,Z 183.573,A 133.371,B 90.000,C 0.000} C_DIS
LIN {X 198.927,Y -211.017,Z 183.615,A 133.311,B 90.000,C 0.000} C_DIS
LIN {X 198.880,Y -211.061,Z 183.666,A 133.298,B 90.000,C 0.000} C_DIS
LIN {X 198.810,Y -211.127,Z 183.717,A 133.279,B 90.000,C 0.000} C_DIS
LIN {X 198.642,Y -211.285,Z 183.738,A 133.233,B 90.000,C 0.000} C_DIS
LIN {X 198.413,Y -211.500,Z 183.693,A 133.171,B 90.000,C 0.000} C_DIS
LIN {X 198.220,Y -211.681,Z 183.488,A 133.119,B 90.000,C 0.000} C_DIS
LIN {X 198.037,Y -211.852,Z 183.237,A 133.070,B 90.000,C 0.000} C_DIS
LIN {X 198.023,Y -211.866,Z 181.923,A 133.066,B 90.000,C 0.000} C_DIS
LIN {X 197.984,Y -211.901,Z 181.715,A 133.055,B 90.000,C 0.000} C_DIS
LIN {X 197.932,Y -211.951,Z 179.216,A 133.041,B 90.000,C 0.000} C_DIS
LIN {X 197.932,Y -211.951,Z 177.156,A 133.041,B 90.000,C 0.000} C_DIS
LIN {X 198.061,Y -211.830,Z 176.979,A 133.076,B 90.000,C 0.000} C_DIS
LIN {X 198.177,Y -211.722,Z 176.853,A 133.107,B 90.000,C 0.000} C_DIS
LIN {X 198.272,Y -211.632,Z 176.801,A 133.133,B 90.000,C 0.000} C_DIS
LIN {X 198.330,Y -211.578,Z 176.780,A 133.149,B 90.000,C 0.000} C_DIS
LIN {X 198.354,Y -211.556,Z 176.729,A 133.155,B 90.000,C 0.000} C_DIS
LIN {X 198.385,Y -211.527,Z 176.678,A 133.164,B 90.000,C 0.000} C_DIS
LIN {X 198.533,Y -211.387,Z 176.635,A 133.204,B 90.000,C 0.000} C_DIS
LIN {X 198.595,Y -211.329,Z 176.533,A 133.221,B 90.000,C 0.000} C_DIS
LIN {X 198.744,Y -211.189,Z 176.491,A 133.261,B 90.000,C 0.000} C_DIS
LIN {X 198.775,Y -211.160,Z 176.440,A 133.270,B 90.000,C 0.000} C_DIS
LIN {X 198.821,Y -211.116,Z 176.389,A 133.282,B 90.000,C 0.000} C_DIS
LIN {X 199.044,Y -210.906,Z 176.346,A 133.343,B 90.000,C 0.000} C_DIS
LIN {X 199.090,Y -210.862,Z 176.295,A 133.355,B 90.000,C 0.000} C_DIS
LIN {X 199.121,Y -210.833,Z 176.244,A 133.364,B 90.000,C 0.000} C_DIS
LIN {X 199.270,Y -210.693,Z 176.202,A 133.404,B 90.000,C 0.000} C_DIS
LIN {X 199.331,Y -210.635,Z 176.100,A 133.421,B 90.000,C 0.000} C_DIS
LIN {X 199.480,Y -210.494,Z 176.057,A 133.461,B 90.000,C 0.000} C_DIS
LIN {X 199.541,Y -210.436,Z 175.955,A 133.478,B 90.000,C 0.000} C_DIS
LIN {X 199.689,Y -210.295,Z 175.913,A 133.518,B 90.000,C 0.000} C_DIS
LIN {X 199.720,Y -210.266,Z 175.862,A 133.527,B 90.000,C 0.000} C_DIS
LIN {X 199.766,Y -210.222,Z 175.811,A 133.539,B 90.000,C 0.000} C_DIS
LIN {X 199.988,Y -210.011,Z 175.768,A 133.600,B 90.000,C 0.000} C_DIS
LIN {X 200.034,Y -209.967,Z 175.717,A 133.612,B 90.000,C 0.000} C_DIS
LIN {X 200.065,Y -209.938,Z 175.666,A 133.621,B 90.000,C 0.000} C_DIS
LIN {X 200.213,Y -209.797,Z 175.624,A 133.661,B 90.000,C 0.000} C_DIS
LIN {X 200.274,Y -209.739,Z 175.522,A 133.678,B 90.000,C 0.000} C_DIS
LIN {X 200.422,Y -209.597,Z 175.479,A 133.718,B 90.000,C 0.000} C_DIS
LIN {X 200.452,Y -209.568,Z 175.428,A 133.726,B 90.000,C 0.000} C_DIS
LIN {X 200.498,Y -209.524,Z 175.377,A 133.739,B 90.000,C 0.000} C_DIS
LIN {X 200.720,Y -209.312,Z 175.335,A 133.799,B 90.000,C 0.000} C_DIS
LIN {X 200.766,Y -209.268,Z 175.284,A 133.812,B 90.000,C 0.000} C_DIS
LIN {X 200.796,Y -209.239,Z 175.233,A 133.820,B 90.000,C 0.000} C_DIS
LIN {X 200.943,Y -209.097,Z 175.190,A 133.861,B 90.000,C 0.000} C_DIS
LIN {X 201.005,Y -209.039,Z 175.088,A 133.878,B 90.000,C 0.000} C_DIS
LIN {X 201.152,Y -208.897,Z 175.046,A 133.918,B 90.000,C 0.000} C_DIS
LIN {X 201.182,Y -208.868,Z 174.995,A 133.926,B 90.000,C 0.000} C_DIS
LIN {X 201.228,Y -208.823,Z 174.944,A 133.939,B 90.000,C 0.000} C_DIS
LIN {X 201.449,Y -208.611,Z 174.901,A 133.999,B 90.000,C 0.000} C_DIS
LIN {X 201.494,Y -208.567,Z 174.850,A 134.012,B 90.000,C 0.000} C_DIS
LIN {X 201.525,Y -208.537,Z 174.799,A 134.020,B 90.000,C 0.000} C_DIS
LIN {X 201.672,Y -208.395,Z 174.757,A 134.061,B 90.000,C 0.000} C_DIS
LIN {X 201.733,Y -208.336,Z 174.654,A 134.077,B 90.000,C 0.000} C_DIS
LIN {X 201.879,Y -208.194,Z 174.612,A 134.118,B 90.000,C 0.000} C_DIS
LIN {X 201.910,Y -208.164,Z 174.561,A 134.126,B 90.000,C 0.000} C_DIS
LIN {X 201.955,Y -208.120,Z 174.510,A 134.139,B 90.000,C 0.000} C_DIS
LIN {X 202.175,Y -207.907,Z 174.467,A 134.199,B 90.000,C 0.000} C_DIS
LIN {X 202.221,Y -207.862,Z 174.416,A 134.212,B 90.000,C 0.000} C_DIS
LIN {X 202.251,Y -207.833,Z 174.365,A 134.220,B 90.000,C 0.000} C_DIS
LIN {X 202.397,Y -207.690,Z 174.323,A 134.261,B 90.000,C 0.000} C_DIS
LIN {X 202.458,Y -207.631,Z 174.221,A 134.277,B 90.000,C 0.000} C_DIS
LIN {X 202.604,Y -207.488,Z 174.178,A 134.318,B 90.000,C 0.000} C_DIS
LIN {X 202.635,Y -207.459,Z 174.127,A 134.326,B 90.000,C 0.000} C_DIS
LIN {X 202.680,Y -207.414,Z 174.076,A 134.339,B 90.000,C 0.000} C_DIS
LIN {X 202.899,Y -207.200,Z 174.034,A 134.399,B 90.000,C 0.000} C_DIS
LIN {X 202.945,Y -207.156,Z 173.983,A 134.412,B 90.000,C 0.000} C_DIS
LIN {X 202.975,Y -207.126,Z 173.932,A 134.420,B 90.000,C 0.000} C_DIS
LIN {X 203.121,Y -206.983,Z 173.889,A 134.460,B 90.000,C 0.000} C_DIS
LIN {X 203.181,Y -206.923,Z 173.787,A 134.477,B 90.000,C 0.000} C_DIS
LIN {X 203.327,Y -206.780,Z 173.745,A 134.518,B 90.000,C 0.000} C_DIS
LIN {X 203.357,Y -206.751,Z 173.694,A 134.526,B 90.000,C 0.000} C_DIS
LIN {X 203.403,Y -206.706,Z 173.643,A 134.539,B 90.000,C 0.000} C_DIS
LIN {X 203.621,Y -206.491,Z 173.600,A 134.599,B 90.000,C 0.000} C_DIS
LIN {X 203.666,Y -206.446,Z 173.549,A 134.612,B 90.000,C 0.000} C_DIS
LIN {X 203.696,Y -206.417,Z 173.498,A 134.620,B 90.000,C 0.000} C_DIS
LIN {X 203.842,Y -206.273,Z 173.456,A 134.660,B 90.000,C 0.000} C_DIS
LIN {X 203.902,Y -206.213,Z 173.354,A 134.677,B 90.000,C 0.000} C_DIS
LIN {X 204.047,Y -206.070,Z 173.311,A 134.717,B 90.000,C 0.000} C_DIS
LIN {X 204.077,Y -206.040,Z 173.260,A 134.726,B 90.000,C 0.000} C_DIS
LIN {X 204.123,Y -205.995,Z 173.209,A 134.738,B 90.000,C 0.000} C_DIS
LIN {X 204.340,Y -205.779,Z 173.167,A 134.799,B 90.000,C 0.000} C_DIS
LIN {X 204.385,Y -205.735,Z 173.116,A 134.811,B 90.000,C 0.000} C_DIS
LIN {X 204.415,Y -205.705,Z 173.065,A 134.820,B 90.000,C 0.000} C_DIS
LIN {X 204.560,Y -205.561,Z 173.022,A 134.860,B 90.000,C 0.000} C_DIS
LIN {X 204.620,Y -205.501,Z 172.920,A 134.877,B 90.000,C 0.000} C_DIS
LIN {X 204.765,Y -205.357,Z 172.878,A 134.917,B 90.000,C 0.000} C_DIS
LIN {X 204.795,Y -205.327,Z 172.827,A 134.926,B 90.000,C 0.000} C_DIS
LIN {X 204.840,Y -205.282,Z 172.776,A 134.938,B 90.000,C 0.000} C_DIS
LIN {X 205.057,Y -205.065,Z 172.733,A 134.999,B 90.000,C 0.000} C_DIS
LIN {X 205.102,Y -205.020,Z 172.682,A 135.011,B 90.000,C 0.000} C_DIS
LIN {X 205.132,Y -204.990,Z 172.631,A 135.020,B 90.000,C 0.000} C_DIS
LIN {X 205.276,Y -204.846,Z 172.589,A 135.060,B 90.000,C 0.000} C_DIS
LIN {X 205.336,Y -204.786,Z 172.487,A 135.077,B 90.000,C 0.000} C_DIS
LIN {X 205.480,Y -204.641,Z 172.444,A 135.117,B 90.000,C 0.000} C_DIS
LIN {X 205.510,Y -204.611,Z 172.393,A 135.126,B 90.000,C 0.000} C_DIS
LIN {X 205.555,Y -204.566,Z 172.342,A 135.138,B 90.000,C 0.000} C_DIS
LIN {X 205.771,Y -204.349,Z 172.300,A 135.199,B 90.000,C 0.000} C_DIS
LIN {X 205.816,Y -204.304,Z 172.249,A 135.211,B 90.000,C 0.000} C_DIS
LIN {X 205.845,Y -204.273,Z 172.197,A 135.220,B 90.000,C 0.000} C_DIS
LIN {X 205.989,Y -204.128,Z 172.155,A 135.260,B 90.000,C 0.000} C_DIS
LIN {X 206.049,Y -204.068,Z 172.053,A 135.277,B 90.000,C 0.000} C_DIS
LIN {X 206.193,Y -203.923,Z 172.010,A 135.317,B 90.000,C 0.000} C_DIS
LIN {X 206.252,Y -203.863,Z 171.908,A 135.334,B 90.000,C 0.000} C_DIS
LIN {X 206.396,Y -203.717,Z 171.866,A 135.374,B 90.000,C 0.000} C_DIS
LIN {X 206.426,Y -203.687,Z 171.815,A 135.383,B 90.000,C 0.000} C_DIS
LIN {X 206.470,Y -203.642,Z 171.764,A 135.395,B 90.000,C 0.000} C_DIS
LIN {X 206.685,Y -203.424,Z 171.721,A 135.456,B 90.000,C 0.000} C_DIS
LIN {X 206.730,Y -203.378,Z 171.670,A 135.468,B 90.000,C 0.000} C_DIS
LIN {X 206.760,Y -203.348,Z 171.619,A 135.477,B 90.000,C 0.000} C_DIS
LIN {X 206.903,Y -203.202,Z 171.577,A 135.517,B 90.000,C 0.000} C_DIS
LIN {X 206.962,Y -203.142,Z 171.475,A 135.534,B 90.000,C 0.000} C_DIS
LIN {X 207.105,Y -202.996,Z 171.432,A 135.574,B 90.000,C 0.000} C_DIS
LIN {X 207.135,Y -202.966,Z 171.381,A 135.582,B 90.000,C 0.000} C_DIS
LIN {X 207.179,Y -202.920,Z 171.330,A 135.595,B 90.000,C 0.000} C_DIS
LIN {X 207.394,Y -202.701,Z 171.288,A 135.656,B 90.000,C 0.000} C_DIS
LIN {X 207.438,Y -202.656,Z 171.237,A 135.668,B 90.000,C 0.000} C_DIS
LIN {X 207.468,Y -202.626,Z 171.186,A 135.677,B 90.000,C 0.000} C_DIS
LIN {X 207.610,Y -202.479,Z 171.143,A 135.717,B 90.000,C 0.000} C_DIS
LIN {X 207.670,Y -202.419,Z 171.041,A 135.734,B 90.000,C 0.000} C_DIS
LIN {X 207.812,Y -202.272,Z 170.999,A 135.774,B 90.000,C 0.000} C_DIS
LIN {X 207.842,Y -202.242,Z 170.948,A 135.782,B 90.000,C 0.000} C_DIS
LIN {X 207.886,Y -202.196,Z 170.897,A 135.795,B 90.000,C 0.000} C_DIS
LIN {X 208.100,Y -201.977,Z 170.854,A 135.855,B 90.000,C 0.000} C_DIS
LIN {X 208.144,Y -201.931,Z 170.803,A 135.868,B 90.000,C 0.000} C_DIS
LIN {X 208.173,Y -201.901,Z 170.752,A 135.876,B 90.000,C 0.000} C_DIS
LIN {X 208.315,Y -201.754,Z 170.710,A 135.917,B 90.000,C 0.000} C_DIS
LIN {X 208.375,Y -201.693,Z 170.608,A 135.933,B 90.000,C 0.000} C_DIS
LIN {X 208.516,Y -201.546,Z 170.565,A 135.974,B 90.000,C 0.000} C_DIS
LIN {X 208.546,Y -201.516,Z 170.514,A 135.982,B 90.000,C 0.000} C_DIS
LIN {X 208.590,Y -201.470,Z 170.463,A 135.995,B 90.000,C 0.000} C_DIS
LIN {X 208.803,Y -201.250,Z 170.421,A 136.055,B 90.000,C 0.000} C_DIS
LIN {X 208.847,Y -201.204,Z 170.370,A 136.068,B 90.000,C 0.000} C_DIS
LIN {X 208.877,Y -201.173,Z 170.319,A 136.076,B 90.000,C 0.000} C_DIS
LIN {X 209.018,Y -201.026,Z 170.276,A 136.117,B 90.000,C 0.000} C_DIS
LIN {X 209.077,Y -200.965,Z 170.174,A 136.133,B 90.000,C 0.000} C_DIS
LIN {X 209.218,Y -200.818,Z 170.132,A 136.174,B 90.000,C 0.000} C_DIS
LIN {X 209.248,Y -200.787,Z 170.081,A 136.182,B 90.000,C 0.000} C_DIS
LIN {X 209.292,Y -200.741,Z 170.030,A 136.195,B 90.000,C 0.000} C_DIS
LIN {X 209.504,Y -200.520,Z 169.987,A 136.255,B 90.000,C 0.000} C_DIS
LIN {X 209.548,Y -200.474,Z 169.936,A 136.268,B 90.000,C 0.000} C_DIS
LIN {X 209.577,Y -200.443,Z 169.885,A 136.276,B 90.000,C 0.000} C_DIS
LIN {X 209.718,Y -200.296,Z 169.843,A 136.316,B 90.000,C 0.000} C_DIS
LIN {X 209.777,Y -200.234,Z 169.740,A 136.333,B 90.000,C 0.000} C_DIS
LIN {X 209.918,Y -200.086,Z 169.698,A 136.374,B 90.000,C 0.000} C_DIS
LIN {X 209.947,Y -200.056,Z 169.647,A 136.382,B 90.000,C 0.000} C_DIS
LIN {X 209.991,Y -200.010,Z 169.596,A 136.395,B 90.000,C 0.000} C_DIS
LIN {X 210.202,Y -199.788,Z 169.554,A 136.455,B 90.000,C 0.000} C_DIS
LIN {X 210.246,Y -199.742,Z 169.502,A 136.468,B 90.000,C 0.000} C_DIS
LIN {X 210.275,Y -199.711,Z 169.451,A 136.476,B 90.000,C 0.000} C_DIS
LIN {X 210.416,Y -199.563,Z 169.409,A 136.516,B 90.000,C 0.000} C_DIS
LIN {X 210.474,Y -199.501,Z 169.307,A 136.533,B 90.000,C 0.000} C_DIS
LIN {X 210.614,Y -199.353,Z 169.264,A 136.573,B 90.000,C 0.000} C_DIS
LIN {X 210.644,Y -199.322,Z 169.213,A 136.582,B 90.000,C 0.000} C_DIS
LIN {X 210.687,Y -199.276,Z 169.162,A 136.594,B 90.000,C 0.000} C_DIS
LIN {X 210.898,Y -199.053,Z 169.120,A 136.655,B 90.000,C 0.000} C_DIS
LIN {X 210.941,Y -199.007,Z 169.069,A 136.668,B 90.000,C 0.000} C_DIS
LIN {X 210.970,Y -198.976,Z 169.018,A 136.676,B 90.000,C 0.000} C_DIS
LIN {X 211.110,Y -198.827,Z 168.975,A 136.716,B 90.000,C 0.000} C_DIS
LIN {X 211.169,Y -198.766,Z 168.873,A 136.733,B 90.000,C 0.000} C_DIS
LIN {X 211.309,Y -198.617,Z 168.831,A 136.773,B 90.000,C 0.000} C_DIS
LIN {X 211.367,Y -198.555,Z 168.729,A 136.790,B 90.000,C 0.000} C_DIS
LIN {X 211.506,Y -198.406,Z 168.686,A 136.830,B 90.000,C 0.000} C_DIS
LIN {X 211.535,Y -198.375,Z 168.635,A 136.839,B 90.000,C 0.000} C_DIS
LIN {X 211.579,Y -198.329,Z 168.584,A 136.851,B 90.000,C 0.000} C_DIS
LIN {X 211.788,Y -198.105,Z 168.542,A 136.912,B 90.000,C 0.000} C_DIS
LIN {X 211.832,Y -198.059,Z 168.491,A 136.925,B 90.000,C 0.000} C_DIS
LIN {X 211.861,Y -198.028,Z 168.440,A 136.933,B 90.000,C 0.000} C_DIS
LIN {X 212.000,Y -197.879,Z 168.397,A 136.973,B 90.000,C 0.000} C_DIS
LIN {X 212.058,Y -197.816,Z 168.295,A 136.990,B 90.000,C 0.000} C_DIS
LIN {X 212.197,Y -197.667,Z 168.253,A 137.030,B 90.000,C 0.000} C_DIS
LIN {X 212.226,Y -197.636,Z 168.202,A 137.039,B 90.000,C 0.000} C_DIS
LIN {X 212.270,Y -197.589,Z 168.151,A 137.051,B 90.000,C 0.000} C_DIS
LIN {X 212.478,Y -197.365,Z 168.108,A 137.112,B 90.000,C 0.000} C_DIS
LIN {X 212.521,Y -197.319,Z 168.057,A 137.124,B 90.000,C 0.000} C_DIS
LIN {X 212.550,Y -197.287,Z 168.006,A 137.133,B 90.000,C 0.000} C_DIS
LIN {X 212.689,Y -197.138,Z 167.964,A 137.173,B 90.000,C 0.000} C_DIS
LIN {X 212.747,Y -197.075,Z 167.862,A 137.190,B 90.000,C 0.000} C_DIS
LIN {X 212.886,Y -196.926,Z 167.819,A 137.230,B 90.000,C 0.000} C_DIS
LIN {X 212.914,Y -196.895,Z 167.768,A 137.239,B 90.000,C 0.000} C_DIS
LIN {X 212.958,Y -196.848,Z 167.717,A 137.251,B 90.000,C 0.000} C_DIS
LIN {X 213.165,Y -196.623,Z 167.675,A 137.312,B 90.000,C 0.000} C_DIS
LIN {X 213.209,Y -196.576,Z 167.624,A 137.324,B 90.000,C 0.000} C_DIS
LIN {X 213.237,Y -196.545,Z 167.573,A 137.333,B 90.000,C 0.000} C_DIS
LIN {X 213.376,Y -196.395,Z 167.530,A 137.373,B 90.000,C 0.000} C_DIS
LIN {X 213.433,Y -196.332,Z 167.428,A 137.390,B 90.000,C 0.000} C_DIS
LIN {X 213.571,Y -196.182,Z 167.386,A 137.430,B 90.000,C 0.000} C_DIS
LIN {X 213.600,Y -196.151,Z 167.335,A 137.439,B 90.000,C 0.000} C_DIS
LIN {X 213.643,Y -196.104,Z 167.284,A 137.451,B 90.000,C 0.000} C_DIS
LIN {X 213.850,Y -195.878,Z 167.241,A 137.512,B 90.000,C 0.000} C_DIS
LIN {X 213.893,Y -195.831,Z 167.190,A 137.524,B 90.000,C 0.000} C_DIS
LIN {X 213.922,Y -195.800,Z 167.139,A 137.533,B 90.000,C 0.000} C_DIS
LIN {X 214.059,Y -195.649,Z 167.097,A 137.573,B 90.000,C 0.000} C_DIS
LIN {X 214.117,Y -195.586,Z 166.994,A 137.590,B 90.000,C 0.000} C_DIS
LIN {X 214.254,Y -195.436,Z 166.952,A 137.630,B 90.000,C 0.000} C_DIS
LIN {X 214.283,Y -195.404,Z 166.901,A 137.638,B 90.000,C 0.000} C_DIS
LIN {X 214.326,Y -195.357,Z 166.850,A 137.651,B 90.000,C 0.000} C_DIS
LIN {X 214.532,Y -195.131,Z 166.807,A 137.711,B 90.000,C 0.000} C_DIS
LIN {X 214.575,Y -195.084,Z 166.756,A 137.724,B 90.000,C 0.000} C_DIS
LIN {X 214.603,Y -195.052,Z 166.705,A 137.732,B 90.000,C 0.000} C_DIS
LIN {X 214.741,Y -194.901,Z 166.663,A 137.773,B 90.000,C 0.000} C_DIS
LIN {X 214.798,Y -194.838,Z 166.561,A 137.790,B 90.000,C 0.000} C_DIS
LIN {X 214.935,Y -194.687,Z 166.518,A 137.830,B 90.000,C 0.000} C_DIS
LIN {X 214.963,Y -194.655,Z 166.467,A 137.838,B 90.000,C 0.000} C_DIS
LIN {X 215.006,Y -194.608,Z 166.416,A 137.851,B 90.000,C 0.000} C_DIS
LIN {X 215.212,Y -194.381,Z 166.374,A 137.911,B 90.000,C 0.000} C_DIS
LIN {X 215.254,Y -194.334,Z 166.323,A 137.924,B 90.000,C 0.000} C_DIS
LIN {X 215.283,Y -194.302,Z 166.272,A 137.932,B 90.000,C 0.000} C_DIS
LIN {X 215.419,Y -194.151,Z 166.229,A 137.973,B 90.000,C 0.000} C_DIS
LIN {X 215.476,Y -194.088,Z 166.127,A 137.989,B 90.000,C 0.000} C_DIS
LIN {X 215.613,Y -193.936,Z 166.085,A 138.030,B 90.000,C 0.000} C_DIS
LIN {X 215.641,Y -193.904,Z 166.034,A 138.038,B 90.000,C 0.000} C_DIS
LIN {X 215.684,Y -193.857,Z 165.983,A 138.051,B 90.000,C 0.000} C_DIS
LIN {X 215.888,Y -193.629,Z 165.940,A 138.111,B 90.000,C 0.000} C_DIS
LIN {X 215.931,Y -193.582,Z 165.889,A 138.124,B 90.000,C 0.000} C_DIS
LIN {X 215.959,Y -193.550,Z 165.838,A 138.132,B 90.000,C 0.000} C_DIS
LIN {X 216.095,Y -193.398,Z 165.796,A 138.173,B 90.000,C 0.000} C_DIS
LIN {X 216.152,Y -193.335,Z 165.694,A 138.189,B 90.000,C 0.000} C_DIS
LIN {X 216.288,Y -193.183,Z 165.651,A 138.230,B 90.000,C 0.000} C_DIS
LIN {X 216.316,Y -193.151,Z 165.600,A 138.238,B 90.000,C 0.000} C_DIS
LIN {X 216.359,Y -193.103,Z 165.549,A 138.251,B 90.000,C 0.000} C_DIS
LIN {X 216.562,Y -192.875,Z 165.507,A 138.311,B 90.000,C 0.000} C_DIS
LIN {X 216.605,Y -192.827,Z 165.456,A 138.324,B 90.000,C 0.000} C_DIS
LIN {X 216.633,Y -192.796,Z 165.405,A 138.332,B 90.000,C 0.000} C_DIS
LIN {X 216.769,Y -192.643,Z 165.362,A 138.372,B 90.000,C 0.000} C_DIS
LIN {X 216.825,Y -192.579,Z 165.260,A 138.389,B 90.000,C 0.000} C_DIS
LIN {X 216.961,Y -192.427,Z 165.218,A 138.430,B 90.000,C 0.000} C_DIS
LIN {X 217.017,Y -192.363,Z 165.116,A 138.446,B 90.000,C 0.000} C_DIS
LIN {X 217.152,Y -192.210,Z 165.073,A 138.487,B 90.000,C 0.000} C_DIS
LIN {X 217.180,Y -192.179,Z 165.022,A 138.495,B 90.000,C 0.000} C_DIS
LIN {X 217.223,Y -192.131,Z 164.971,A 138.508,B 90.000,C 0.000} C_DIS
LIN {X 217.425,Y -191.901,Z 164.929,A 138.568,B 90.000,C 0.000} C_DIS
LIN {X 217.468,Y -191.854,Z 164.878,A 138.581,B 90.000,C 0.000} C_DIS
LIN {X 217.496,Y -191.822,Z 164.827,A 138.589,B 90.000,C 0.000} C_DIS
LIN {X 217.631,Y -191.669,Z 164.784,A 138.629,B 90.000,C 0.000} C_DIS
LIN {X 217.687,Y -191.605,Z 164.682,A 138.646,B 90.000,C 0.000} C_DIS
LIN {X 217.822,Y -191.452,Z 164.640,A 138.687,B 90.000,C 0.000} C_DIS
LIN {X 217.850,Y -191.420,Z 164.589,A 138.695,B 90.000,C 0.000} C_DIS
LIN {X 217.892,Y -191.372,Z 164.537,A 138.707,B 90.000,C 0.000} C_DIS
LIN {X 218.094,Y -191.142,Z 164.495,A 138.768,B 90.000,C 0.000} C_DIS
LIN {X 218.136,Y -191.094,Z 164.444,A 138.781,B 90.000,C 0.000} C_DIS
LIN {X 218.164,Y -191.062,Z 164.393,A 138.789,B 90.000,C 0.000} C_DIS
LIN {X 218.298,Y -190.908,Z 164.350,A 138.829,B 90.000,C 0.000} C_DIS
LIN {X 218.354,Y -190.844,Z 164.248,A 138.846,B 90.000,C 0.000} C_DIS
LIN {X 218.488,Y -190.691,Z 164.206,A 138.886,B 90.000,C 0.000} C_DIS
LIN {X 218.516,Y -190.659,Z 164.155,A 138.895,B 90.000,C 0.000} C_DIS
LIN {X 218.558,Y -190.611,Z 164.104,A 138.907,B 90.000,C 0.000} C_DIS
LIN {X 218.759,Y -190.380,Z 164.061,A 138.968,B 90.000,C 0.000} C_DIS
LIN {X 218.801,Y -190.332,Z 164.010,A 138.980,B 90.000,C 0.000} C_DIS
LIN {X 218.829,Y -190.300,Z 163.959,A 138.989,B 90.000,C 0.000} C_DIS
LIN {X 218.963,Y -190.146,Z 163.917,A 139.029,B 90.000,C 0.000} C_DIS
LIN {X 219.018,Y -190.082,Z 163.815,A 139.046,B 90.000,C 0.000} C_DIS
LIN {X 219.152,Y -189.927,Z 163.772,A 139.086,B 90.000,C 0.000} C_DIS
LIN {X 219.180,Y -189.895,Z 163.721,A 139.095,B 90.000,C 0.000} C_DIS
LIN {X 219.222,Y -189.847,Z 163.670,A 139.107,B 90.000,C 0.000} C_DIS
LIN {X 219.422,Y -189.615,Z 163.628,A 139.168,B 90.000,C 0.000} C_DIS
LIN {X 219.464,Y -189.567,Z 163.577,A 139.180,B 90.000,C 0.000} C_DIS
LIN {X 219.491,Y -189.535,Z 163.526,A 139.189,B 90.000,C 0.000} C_DIS
LIN {X 219.625,Y -189.381,Z 163.483,A 139.229,B 90.000,C 0.000} C_DIS
LIN {X 219.680,Y -189.316,Z 163.381,A 139.246,B 90.000,C 0.000} C_DIS
LIN {X 219.813,Y -189.162,Z 163.339,A 139.286,B 90.000,C 0.000} C_DIS
LIN {X 219.841,Y -189.129,Z 163.288,A 139.295,B 90.000,C 0.000} C_DIS
LIN {X 219.883,Y -189.081,Z 163.237,A 139.307,B 90.000,C 0.000} C_DIS
LIN {X 220.082,Y -188.849,Z 163.194,A 139.368,B 90.000,C 0.000} C_DIS
LIN {X 220.124,Y -188.801,Z 163.143,A 139.380,B 90.000,C 0.000} C_DIS
LIN {X 220.151,Y -188.768,Z 163.092,A 139.389,B 90.000,C 0.000} C_DIS
LIN {X 220.284,Y -188.613,Z 163.050,A 139.429,B 90.000,C 0.000} C_DIS
LIN {X 220.339,Y -188.549,Z 162.948,A 139.446,B 90.000,C 0.000} C_DIS
LIN {X 220.472,Y -188.394,Z 162.905,A 139.486,B 90.000,C 0.000} C_DIS
LIN {X 220.499,Y -188.361,Z 162.854,A 139.494,B 90.000,C 0.000} C_DIS
LIN {X 220.541,Y -188.313,Z 162.803,A 139.507,B 90.000,C 0.000} C_DIS
LIN {X 220.740,Y -188.080,Z 162.761,A 139.568,B 90.000,C 0.000} C_DIS
LIN {X 220.781,Y -188.031,Z 162.710,A 139.580,B 90.000,C 0.000} C_DIS
LIN {X 220.808,Y -187.999,Z 162.659,A 139.588,B 90.000,C 0.000} C_DIS
LIN {X 220.941,Y -187.844,Z 162.616,A 139.629,B 90.000,C 0.000} C_DIS
LIN {X 220.996,Y -187.779,Z 162.514,A 139.646,B 90.000,C 0.000} C_DIS
LIN {X 221.128,Y -187.623,Z 162.472,A 139.686,B 90.000,C 0.000} C_DIS
LIN {X 221.155,Y -187.591,Z 162.421,A 139.694,B 90.000,C 0.000} C_DIS
LIN {X 221.196,Y -187.542,Z 162.370,A 139.707,B 90.000,C 0.000} C_DIS
LIN {X 221.394,Y -187.309,Z 162.327,A 139.767,B 90.000,C 0.000} C_DIS
LIN {X 221.435,Y -187.260,Z 162.276,A 139.780,B 90.000,C 0.000} C_DIS
LIN {X 221.463,Y -187.228,Z 162.225,A 139.788,B 90.000,C 0.000} C_DIS
LIN {X 221.595,Y -187.072,Z 162.183,A 139.829,B 90.000,C 0.000} C_DIS
LIN {X 221.649,Y -187.007,Z 162.080,A 139.845,B 90.000,C 0.000} C_DIS
LIN {X 221.781,Y -186.851,Z 162.038,A 139.886,B 90.000,C 0.000} C_DIS
LIN {X 221.836,Y -186.786,Z 161.936,A 139.903,B 90.000,C 0.000} C_DIS
LIN {X 221.967,Y -186.630,Z 161.894,A 139.943,B 90.000,C 0.000} C_DIS
LIN {X 221.994,Y -186.597,Z 161.842,A 139.951,B 90.000,C 0.000} C_DIS
LIN {X 222.035,Y -186.548,Z 161.791,A 139.964,B 90.000,C 0.000} C_DIS
LIN {X 222.232,Y -186.314,Z 161.749,A 140.024,B 90.000,C 0.000} C_DIS
LIN {X 222.273,Y -186.265,Z 161.698,A 140.037,B 90.000,C 0.000} C_DIS
LIN {X 222.300,Y -186.232,Z 161.647,A 140.045,B 90.000,C 0.000} C_DIS
LIN {X 222.431,Y -186.076,Z 161.604,A 140.086,B 90.000,C 0.000} C_DIS
LIN {X 222.486,Y -186.011,Z 161.502,A 140.102,B 90.000,C 0.000} C_DIS
LIN {X 222.617,Y -185.854,Z 161.460,A 140.143,B 90.000,C 0.000} C_DIS
LIN {X 222.644,Y -185.822,Z 161.409,A 140.151,B 90.000,C 0.000} C_DIS
LIN {X 222.685,Y -185.773,Z 161.358,A 140.164,B 90.000,C 0.000} C_DIS
LIN {X 222.881,Y -185.537,Z 161.315,A 140.224,B 90.000,C 0.000} C_DIS
LIN {X 222.922,Y -185.488,Z 161.264,A 140.237,B 90.000,C 0.000} C_DIS
LIN {X 222.949,Y -185.456,Z 161.213,A 140.245,B 90.000,C 0.000} C_DIS
LIN {X 223.079,Y -185.299,Z 161.171,A 140.286,B 90.000,C 0.000} C_DIS
LIN {X 223.134,Y -185.233,Z 161.069,A 140.302,B 90.000,C 0.000} C_DIS
LIN {X 223.264,Y -185.076,Z 161.026,A 140.343,B 90.000,C 0.000} C_DIS
LIN {X 223.291,Y -185.044,Z 160.975,A 140.351,B 90.000,C 0.000} C_DIS
LIN {X 223.332,Y -184.995,Z 160.924,A 140.364,B 90.000,C 0.000} C_DIS
LIN {X 223.527,Y -184.759,Z 160.882,A 140.424,B 90.000,C 0.000} C_DIS
LIN {X 223.567,Y -184.710,Z 160.831,A 140.437,B 90.000,C 0.000} C_DIS
LIN {X 223.594,Y -184.677,Z 160.780,A 140.445,B 90.000,C 0.000} C_DIS
LIN {X 223.724,Y -184.519,Z 160.737,A 140.485,B 90.000,C 0.000} C_DIS
LIN {X 223.778,Y -184.454,Z 160.635,A 140.502,B 90.000,C 0.000} C_DIS
LIN {X 223.908,Y -184.296,Z 160.593,A 140.543,B 90.000,C 0.000} C_DIS
LIN {X 223.935,Y -184.264,Z 160.542,A 140.551,B 90.000,C 0.000} C_DIS
LIN {X 223.976,Y -184.214,Z 160.491,A 140.564,B 90.000,C 0.000} C_DIS
LIN {X 224.170,Y -183.978,Z 160.448,A 140.624,B 90.000,C 0.000} C_DIS
LIN {X 224.210,Y -183.929,Z 160.397,A 140.637,B 90.000,C 0.000} C_DIS
LIN {X 224.237,Y -183.896,Z 160.346,A 140.645,B 90.000,C 0.000} C_DIS
LIN {X 224.367,Y -183.738,Z 160.304,A 140.685,B 90.000,C 0.000} C_DIS
LIN {X 224.420,Y -183.672,Z 160.202,A 140.702,B 90.000,C 0.000} C_DIS
LIN {X 224.550,Y -183.514,Z 160.159,A 140.742,B 90.000,C 0.000} C_DIS
LIN {X 224.577,Y -183.481,Z 160.108,A 140.751,B 90.000,C 0.000} C_DIS
LIN {X 224.617,Y -183.432,Z 160.057,A 140.763,B 90.000,C 0.000} C_DIS
LIN {X 224.810,Y -183.195,Z 160.015,A 140.824,B 90.000,C 0.000} C_DIS
LIN {X 224.851,Y -183.145,Z 159.964,A 140.837,B 90.000,C 0.000} C_DIS
LIN {X 224.877,Y -183.112,Z 159.913,A 140.845,B 90.000,C 0.000} C_DIS
LIN {X 225.006,Y -182.954,Z 159.870,A 140.885,B 90.000,C 0.000} C_DIS
LIN {X 225.060,Y -182.888,Z 159.768,A 140.902,B 90.000,C 0.000} C_DIS
LIN {X 225.189,Y -182.730,Z 159.726,A 140.942,B 90.000,C 0.000} C_DIS
LIN {X 225.242,Y -182.664,Z 159.624,A 140.959,B 90.000,C 0.000} C_DIS
LIN {X 225.371,Y -182.505,Z 159.581,A 140.999,B 90.000,C 0.000} C_DIS
LIN {X 225.397,Y -182.472,Z 159.530,A 141.008,B 90.000,C 0.000} C_DIS
LIN {X 225.437,Y -182.423,Z 159.479,A 141.020,B 90.000,C 0.000} C_DIS
LIN {X 225.630,Y -182.184,Z 159.437,A 141.081,B 90.000,C 0.000} C_DIS
LIN {X 225.670,Y -182.135,Z 159.385,A 141.094,B 90.000,C 0.000} C_DIS
LIN {X 225.697,Y -182.102,Z 159.334,A 141.102,B 90.000,C 0.000} C_DIS
LIN {X 225.825,Y -181.943,Z 159.292,A 141.142,B 90.000,C 0.000} C_DIS
LIN {X 225.851,Y -181.910,Z 159.241,A 141.151,B 90.000,C 0.000} C_DIS
LIN {X 225.891,Y -181.860,Z 159.190,A 141.163,B 90.000,C 0.000} C_DIS
LIN {X 226.083,Y -181.622,Z 159.147,A 141.224,B 90.000,C 0.000} C_DIS
LIN {X 226.123,Y -181.572,Z 159.096,A 141.236,B 90.000,C 0.000} C_DIS
LIN {X 226.150,Y -181.539,Z 159.045,A 141.245,B 90.000,C 0.000} C_DIS
LIN {X 226.277,Y -181.380,Z 159.003,A 141.285,B 90.000,C 0.000} C_DIS
LIN {X 226.330,Y -181.313,Z 158.901,A 141.302,B 90.000,C 0.000} C_DIS
LIN {X 226.458,Y -181.154,Z 158.858,A 141.342,B 90.000,C 0.000} C_DIS
LIN {X 226.511,Y -181.088,Z 158.756,A 141.359,B 90.000,C 0.000} C_DIS
LIN {X 226.638,Y -180.928,Z 158.714,A 141.399,B 90.000,C 0.000} C_DIS
LIN {X 226.665,Y -180.895,Z 158.663,A 141.408,B 90.000,C 0.000} C_DIS
LIN {X 226.705,Y -180.845,Z 158.612,A 141.420,B 90.000,C 0.000} C_DIS
LIN {X 226.896,Y -180.606,Z 158.569,A 141.481,B 90.000,C 0.000} C_DIS
LIN {X 226.935,Y -180.556,Z 158.518,A 141.493,B 90.000,C 0.000} C_DIS
LIN {X 226.962,Y -180.523,Z 158.467,A 141.502,B 90.000,C 0.000} C_DIS
LIN {X 227.089,Y -180.363,Z 158.425,A 141.542,B 90.000,C 0.000} C_DIS
LIN {X 227.141,Y -180.296,Z 158.323,A 141.559,B 90.000,C 0.000} C_DIS
LIN {X 227.268,Y -180.136,Z 158.280,A 141.599,B 90.000,C 0.000} C_DIS
LIN {X 227.295,Y -180.103,Z 158.229,A 141.607,B 90.000,C 0.000} C_DIS
LIN {X 227.334,Y -180.053,Z 158.178,A 141.620,B 90.000,C 0.000} C_DIS
LIN {X 227.524,Y -179.813,Z 158.136,A 141.681,B 90.000,C 0.000} C_DIS
LIN {X 227.564,Y -179.763,Z 158.085,A 141.693,B 90.000,C 0.000} C_DIS
LIN {X 227.590,Y -179.730,Z 158.034,A 141.702,B 90.000,C 0.000} C_DIS
LIN {X 227.716,Y -179.570,Z 157.991,A 141.742,B 90.000,C 0.000} C_DIS
LIN {X 227.769,Y -179.503,Z 157.889,A 141.759,B 90.000,C 0.000} C_DIS
LIN {X 227.895,Y -179.342,Z 157.847,A 141.799,B 90.000,C 0.000} C_DIS
LIN {X 227.922,Y -179.309,Z 157.796,A 141.807,B 90.000,C 0.000} C_DIS
LIN {X 227.961,Y -179.259,Z 157.745,A 141.820,B 90.000,C 0.000} C_DIS
LIN {X 228.150,Y -179.018,Z 157.702,A 141.880,B 90.000,C 0.000} C_DIS
LIN {X 228.189,Y -178.968,Z 157.651,A 141.893,B 90.000,C 0.000} C_DIS
LIN {X 228.216,Y -178.935,Z 157.600,A 141.901,B 90.000,C 0.000} C_DIS
LIN {X 228.342,Y -178.774,Z 157.558,A 141.942,B 90.000,C 0.000} C_DIS
LIN {X 228.394,Y -178.707,Z 157.456,A 141.959,B 90.000,C 0.000} C_DIS
LIN {X 228.520,Y -178.546,Z 157.413,A 141.999,B 90.000,C 0.000} C_DIS
LIN {X 228.546,Y -178.513,Z 157.362,A 142.007,B 90.000,C 0.000} C_DIS
LIN {X 228.585,Y -178.463,Z 157.311,A 142.020,B 90.000,C 0.000} C_DIS
LIN {X 228.773,Y -178.221,Z 157.269,A 142.080,B 90.000,C 0.000} C_DIS
LIN {X 228.812,Y -178.171,Z 157.218,A 142.093,B 90.000,C 0.000} C_DIS
LIN {X 228.838,Y -178.137,Z 157.167,A 142.101,B 90.000,C 0.000} C_DIS
LIN {X 228.964,Y -177.976,Z 157.124,A 142.142,B 90.000,C 0.000} C_DIS
LIN {X 229.016,Y -177.909,Z 157.022,A 142.158,B 90.000,C 0.000} C_DIS
LIN {X 229.141,Y -177.748,Z 156.980,A 142.199,B 90.000,C 0.000} C_DIS
LIN {X 229.167,Y -177.715,Z 156.929,A 142.207,B 90.000,C 0.000} C_DIS
LIN {X 229.206,Y -177.664,Z 156.877,A 142.220,B 90.000,C 0.000} C_DIS
LIN {X 229.394,Y -177.422,Z 156.835,A 142.280,B 90.000,C 0.000} C_DIS
LIN {X 229.433,Y -177.372,Z 156.784,A 142.293,B 90.000,C 0.000} C_DIS
LIN {X 229.459,Y -177.338,Z 156.733,A 142.301,B 90.000,C 0.000} C_DIS
LIN {X 229.583,Y -177.177,Z 156.691,A 142.342,B 90.000,C 0.000} C_DIS
LIN {X 229.635,Y -177.109,Z 156.588,A 142.358,B 90.000,C 0.000} C_DIS
LIN {X 229.760,Y -176.948,Z 156.546,A 142.399,B 90.000,C 0.000} C_DIS
LIN {X 229.786,Y -176.914,Z 156.495,A 142.407,B 90.000,C 0.000} C_DIS
LIN {X 229.825,Y -176.863,Z 156.444,A 142.420,B 90.000,C 0.000} C_DIS
LIN {X 230.011,Y -176.621,Z 156.401,A 142.480,B 90.000,C 0.000} C_DIS
LIN {X 230.050,Y -176.570,Z 156.350,A 142.493,B 90.000,C 0.000} C_DIS
LIN {X 230.076,Y -176.537,Z 156.299,A 142.501,B 90.000,C 0.000} C_DIS
LIN {X 230.200,Y -176.375,Z 156.257,A 142.541,B 90.000,C 0.000} C_DIS
LIN {X 230.252,Y -176.307,Z 156.155,A 142.558,B 90.000,C 0.000} C_DIS
LIN {X 230.376,Y -176.145,Z 156.112,A 142.599,B 90.000,C 0.000} C_DIS
LIN {X 230.401,Y -176.111,Z 156.061,A 142.607,B 90.000,C 0.000} C_DIS
LIN {X 230.440,Y -176.061,Z 156.010,A 142.619,B 90.000,C 0.000} C_DIS
LIN {X 230.626,Y -175.817,Z 155.968,A 142.680,B 90.000,C 0.000} C_DIS
LIN {X 230.665,Y -175.767,Z 155.917,A 142.693,B 90.000,C 0.000} C_DIS
LIN {X 230.690,Y -175.733,Z 155.866,A 142.701,B 90.000,C 0.000} C_DIS
LIN {X 230.814,Y -175.570,Z 155.823,A 142.741,B 90.000,C 0.000} C_DIS
LIN {X 230.865,Y -175.503,Z 155.721,A 142.758,B 90.000,C 0.000} C_DIS
LIN {X 230.989,Y -175.340,Z 155.679,A 142.798,B 90.000,C 0.000} C_DIS
LIN {X 231.014,Y -175.306,Z 155.628,A 142.807,B 90.000,C 0.000} C_DIS
LIN {X 231.053,Y -175.256,Z 155.577,A 142.819,B 90.000,C 0.000} C_DIS
LIN {X 231.238,Y -175.012,Z 155.534,A 142.880,B 90.000,C 0.000} C_DIS
LIN {X 231.276,Y -174.961,Z 155.483,A 142.892,B 90.000,C 0.000} C_DIS
LIN {X 231.302,Y -174.927,Z 155.432,A 142.901,B 90.000,C 0.000} C_DIS
LIN {X 231.425,Y -174.764,Z 155.390,A 142.941,B 90.000,C 0.000} C_DIS
LIN {X 231.476,Y -174.696,Z 155.288,A 142.958,B 90.000,C 0.000} C_DIS
LIN {X 231.599,Y -174.533,Z 155.245,A 142.998,B 90.000,C 0.000} C_DIS
LIN {X 231.650,Y -174.465,Z 155.143,A 143.015,B 90.000,C 0.000} C_DIS
LIN {X 231.773,Y -174.302,Z 155.101,A 143.055,B 90.000,C 0.000} C_DIS
LIN {X 231.798,Y -174.268,Z 155.050,A 143.064,B 90.000,C 0.000} C_DIS
LIN {X 231.837,Y -174.218,Z 154.999,A 143.076,B 90.000,C 0.000} C_DIS
LIN {X 232.021,Y -173.973,Z 154.956,A 143.137,B 90.000,C 0.000} C_DIS
LIN {X 232.059,Y -173.922,Z 154.905,A 143.149,B 90.000,C 0.000} C_DIS
LIN {X 232.084,Y -173.888,Z 154.854,A 143.158,B 90.000,C 0.000} C_DIS
LIN {X 232.207,Y -173.724,Z 154.812,A 143.198,B 90.000,C 0.000} C_DIS
LIN {X 232.257,Y -173.656,Z 154.710,A 143.215,B 90.000,C 0.000} C_DIS
LIN {X 232.380,Y -173.493,Z 154.667,A 143.255,B 90.000,C 0.000} C_DIS
LIN {X 232.405,Y -173.459,Z 154.616,A 143.264,B 90.000,C 0.000} C_DIS
LIN {X 232.443,Y -173.408,Z 154.565,A 143.276,B 90.000,C 0.000} C_DIS
LIN {X 232.626,Y -173.162,Z 154.523,A 143.337,B 90.000,C 0.000} C_DIS
LIN {X 232.664,Y -173.111,Z 154.472,A 143.349,B 90.000,C 0.000} C_DIS
LIN {X 232.689,Y -173.077,Z 154.421,A 143.358,B 90.000,C 0.000} C_DIS
LIN {X 232.811,Y -172.913,Z 154.378,A 143.398,B 90.000,C 0.000} C_DIS
LIN {X 232.862,Y -172.845,Z 154.276,A 143.415,B 90.000,C 0.000} C_DIS
LIN {X 232.983,Y -172.681,Z 154.234,A 143.455,B 90.000,C 0.000} C_DIS
LIN {X 233.009,Y -172.647,Z 154.182,A 143.464,B 90.000,C 0.000} C_DIS
LIN {X 233.047,Y -172.596,Z 154.131,A 143.476,B 90.000,C 0.000} C_DIS
LIN {X 233.229,Y -172.350,Z 154.089,A 143.537,B 90.000,C 0.000} C_DIS
LIN {X 233.267,Y -172.298,Z 154.038,A 143.549,B 90.000,C 0.000} C_DIS
LIN {X 233.292,Y -172.264,Z 153.987,A 143.558,B 90.000,C 0.000} C_DIS
LIN {X 233.413,Y -172.100,Z 153.944,A 143.598,B 90.000,C 0.000} C_DIS
LIN {X 233.463,Y -172.032,Z 153.842,A 143.615,B 90.000,C 0.000} C_DIS
LIN {X 233.584,Y -171.867,Z 153.800,A 143.655,B 90.000,C 0.000} C_DIS
LIN {X 233.610,Y -171.833,Z 153.749,A 143.663,B 90.000,C 0.000} C_DIS
LIN {X 233.647,Y -171.782,Z 153.698,A 143.676,B 90.000,C 0.000} C_DIS
LIN {X 233.829,Y -171.535,Z 153.655,A 143.737,B 90.000,C 0.000} C_DIS
LIN {X 233.866,Y -171.484,Z 153.604,A 143.749,B 90.000,C 0.000} C_DIS
LIN {X 233.891,Y -171.449,Z 153.553,A 143.757,B 90.000,C 0.000} C_DIS
LIN {X 234.012,Y -171.285,Z 153.511,A 143.798,B 90.000,C 0.000} C_DIS
LIN {X 234.062,Y -171.216,Z 153.409,A 143.815,B 90.000,C 0.000} C_DIS
LIN {X 234.183,Y -171.051,Z 153.366,A 143.855,B 90.000,C 0.000} C_DIS
LIN {X 234.208,Y -171.017,Z 153.315,A 143.863,B 90.000,C 0.000} C_DIS
LIN {X 234.245,Y -170.966,Z 153.264,A 143.876,B 90.000,C 0.000} C_DIS
LIN {X 234.426,Y -170.718,Z 153.222,A 143.936,B 90.000,C 0.000} C_DIS
LIN {X 234.463,Y -170.667,Z 153.171,A 143.949,B 90.000,C 0.000} C_DIS
LIN {X 234.488,Y -170.632,Z 153.120,A 143.957,B 90.000,C 0.000} C_DIS
LIN {X 234.608,Y -170.467,Z 153.077,A 143.998,B 90.000,C 0.000} C_DIS
LIN {X 234.658,Y -170.398,Z 152.975,A 144.014,B 90.000,C 0.000} C_DIS
LIN {X 234.778,Y -170.233,Z 152.933,A 144.055,B 90.000,C 0.000} C_DIS
LIN {X 234.803,Y -170.199,Z 152.882,A 144.063,B 90.000,C 0.000} C_DIS
LIN {X 234.840,Y -170.147,Z 152.831,A 144.076,B 90.000,C 0.000} C_DIS
LIN {X 235.020,Y -169.899,Z 152.788,A 144.136,B 90.000,C 0.000} C_DIS
LIN {X 235.057,Y -169.848,Z 152.737,A 144.149,B 90.000,C 0.000} C_DIS
LIN {X 235.082,Y -169.813,Z 152.686,A 144.157,B 90.000,C 0.000} C_DIS
LIN {X 235.201,Y -169.648,Z 152.644,A 144.198,B 90.000,C 0.000} C_DIS
LIN {X 235.251,Y -169.579,Z 152.542,A 144.214,B 90.000,C 0.000} C_DIS
LIN {X 235.370,Y -169.413,Z 152.499,A 144.255,B 90.000,C 0.000} C_DIS
LIN {X 235.395,Y -169.379,Z 152.448,A 144.263,B 90.000,C 0.000} C_DIS
LIN {X 235.432,Y -169.327,Z 152.397,A 144.276,B 90.000,C 0.000} C_DIS
LIN {X 235.611,Y -169.078,Z 152.355,A 144.336,B 90.000,C 0.000} C_DIS
LIN {X 235.648,Y -169.027,Z 152.304,A 144.349,B 90.000,C 0.000} C_DIS
LIN {X 235.673,Y -168.992,Z 152.253,A 144.357,B 90.000,C 0.000} C_DIS
LIN {X 235.792,Y -168.826,Z 152.210,A 144.397,B 90.000,C 0.000} C_DIS
LIN {X 235.841,Y -168.757,Z 152.108,A 144.414,B 90.000,C 0.000} C_DIS
LIN {X 235.960,Y -168.591,Z 152.066,A 144.455,B 90.000,C 0.000} C_DIS
LIN {X 236.009,Y -168.522,Z 151.964,A 144.471,B 90.000,C 0.000} C_DIS
LIN {X 236.128,Y -168.356,Z 151.921,A 144.512,B 90.000,C 0.000} C_DIS
LIN {X 236.152,Y -168.321,Z 151.870,A 144.520,B 90.000,C 0.000} C_DIS
LIN {X 236.189,Y -168.269,Z 151.819,A 144.533,B 90.000,C 0.000} C_DIS
LIN {X 236.367,Y -168.020,Z 151.777,A 144.593,B 90.000,C 0.000} C_DIS
LIN {X 236.404,Y -167.968,Z 151.726,A 144.606,B 90.000,C 0.000} C_DIS
LIN {X 236.428,Y -167.933,Z 151.674,A 144.614,B 90.000,C 0.000} C_DIS
LIN {X 236.547,Y -167.767,Z 151.632,A 144.654,B 90.000,C 0.000} C_DIS
LIN {X 236.596,Y -167.698,Z 151.530,A 144.671,B 90.000,C 0.000} C_DIS
LIN {X 236.714,Y -167.531,Z 151.487,A 144.712,B 90.000,C 0.000} C_DIS
LIN {X 236.738,Y -167.496,Z 151.436,A 144.720,B 90.000,C 0.000} C_DIS
LIN {X 236.775,Y -167.444,Z 151.385,A 144.733,B 90.000,C 0.000} C_DIS
LIN {X 236.952,Y -167.194,Z 151.343,A 144.793,B 90.000,C 0.000} C_DIS
LIN {X 236.988,Y -167.142,Z 151.292,A 144.806,B 90.000,C 0.000} C_DIS
LIN {X 237.013,Y -167.107,Z 151.241,A 144.814,B 90.000,C 0.000} C_DIS
LIN {X 237.130,Y -166.941,Z 151.198,A 144.854,B 90.000,C 0.000} C_DIS
LIN {X 237.179,Y -166.871,Z 151.096,A 144.871,B 90.000,C 0.000} C_DIS
LIN {X 237.297,Y -166.704,Z 151.054,A 144.911,B 90.000,C 0.000} C_DIS
LIN {X 237.321,Y -166.669,Z 151.003,A 144.920,B 90.000,C 0.000} C_DIS
LIN {X 237.358,Y -166.617,Z 150.952,A 144.932,B 90.000,C 0.000} C_DIS
LIN {X 237.534,Y -166.367,Z 150.909,A 144.993,B 90.000,C 0.000} C_DIS
LIN {X 237.570,Y -166.314,Z 150.858,A 145.005,B 90.000,C 0.000} C_DIS
LIN {X 237.594,Y -166.280,Z 150.807,A 145.014,B 90.000,C 0.000} C_DIS
LIN {X 237.711,Y -166.112,Z 150.765,A 145.054,B 90.000,C 0.000} C_DIS
LIN {X 237.760,Y -166.043,Z 150.663,A 145.071,B 90.000,C 0.000} C_DIS
LIN {X 237.877,Y -165.875,Z 150.620,A 145.111,B 90.000,C 0.000} C_DIS
LIN {X 237.901,Y -165.840,Z 150.569,A 145.120,B 90.000,C 0.000} C_DIS
LIN {X 237.938,Y -165.788,Z 150.518,A 145.132,B 90.000,C 0.000} C_DIS
LIN {X 238.112,Y -165.537,Z 150.476,A 145.193,B 90.000,C 0.000} C_DIS
LIN {X 238.149,Y -165.485,Z 150.425,A 145.205,B 90.000,C 0.000} C_DIS
LIN {X 238.173,Y -165.450,Z 150.374,A 145.214,B 90.000,C 0.000} C_DIS
LIN {X 238.289,Y -165.282,Z 150.331,A 145.254,B 90.000,C 0.000} C_DIS
LIN {X 238.338,Y -165.212,Z 150.229,A 145.271,B 90.000,C 0.000} C_DIS
LIN {X 238.454,Y -165.044,Z 150.187,A 145.311,B 90.000,C 0.000} C_DIS
LIN {X 238.478,Y -165.010,Z 150.136,A 145.320,B 90.000,C 0.000} C_DIS
LIN {X 238.514,Y -164.957,Z 150.085,A 145.332,B 90.000,C 0.000} C_DIS
LIN {X 238.689,Y -164.705,Z 150.042,A 145.393,B 90.000,C 0.000} C_DIS
LIN {X 238.725,Y -164.653,Z 149.991,A 145.405,B 90.000,C 0.000} C_DIS
LIN {X 238.749,Y -164.618,Z 149.940,A 145.414,B 90.000,C 0.000} C_DIS
LIN {X 238.865,Y -164.450,Z 149.898,A 145.454,B 90.000,C 0.000} C_DIS
LIN {X 238.913,Y -164.380,Z 149.796,A 145.471,B 90.000,C 0.000} C_DIS
LIN {X 239.028,Y -164.212,Z 149.753,A 145.511,B 90.000,C 0.000} C_DIS
LIN {X 239.052,Y -164.177,Z 149.702,A 145.519,B 90.000,C 0.000} C_DIS
LIN {X 239.088,Y -164.124,Z 149.651,A 145.532,B 90.000,C 0.000} C_DIS
LIN {X 239.262,Y -163.871,Z 149.609,A 145.593,B 90.000,C 0.000} C_DIS
LIN {X 239.298,Y -163.819,Z 149.558,A 145.605,B 90.000,C 0.000} C_DIS
LIN {X 239.322,Y -163.784,Z 149.507,A 145.614,B 90.000,C 0.000} C_DIS
LIN {X 239.437,Y -163.615,Z 149.464,A 145.654,B 90.000,C 0.000} C_DIS
LIN {X 239.485,Y -163.545,Z 149.362,A 145.671,B 90.000,C 0.000} C_DIS
LIN {X 239.600,Y -163.377,Z 149.320,A 145.711,B 90.000,C 0.000} C_DIS
LIN {X 239.624,Y -163.342,Z 149.269,A 145.719,B 90.000,C 0.000} C_DIS
LIN {X 239.660,Y -163.289,Z 149.217,A 145.732,B 90.000,C 0.000} C_DIS
LIN {X 239.832,Y -163.036,Z 149.175,A 145.792,B 90.000,C 0.000} C_DIS
LIN {X 239.868,Y -162.983,Z 149.124,A 145.805,B 90.000,C 0.000} C_DIS
LIN {X 239.892,Y -162.948,Z 149.073,A 145.813,B 90.000,C 0.000} C_DIS
LIN {X 240.006,Y -162.779,Z 149.031,A 145.854,B 90.000,C 0.000} C_DIS
LIN {X 240.054,Y -162.709,Z 148.928,A 145.871,B 90.000,C 0.000} C_DIS
LIN {X 240.168,Y -162.540,Z 148.886,A 145.911,B 90.000,C 0.000} C_DIS
LIN {X 240.216,Y -162.469,Z 148.784,A 145.928,B 90.000,C 0.000} C_DIS
LIN {X 240.330,Y -162.300,Z 148.741,A 145.968,B 90.000,C 0.000} C_DIS
LIN {X 240.354,Y -162.265,Z 148.690,A 145.976,B 90.000,C 0.000} C_DIS
LIN {X 240.390,Y -162.212,Z 148.639,A 145.989,B 90.000,C 0.000} C_DIS
LIN {X 240.561,Y -161.958,Z 148.597,A 146.049,B 90.000,C 0.000} C_DIS
LIN {X 240.596,Y -161.906,Z 148.546,A 146.062,B 90.000,C 0.000} C_DIS
LIN {X 240.620,Y -161.870,Z 148.495,A 146.070,B 90.000,C 0.000} C_DIS
LIN {X 240.734,Y -161.701,Z 148.452,A 146.111,B 90.000,C 0.000} C_DIS
LIN {X 240.781,Y -161.630,Z 148.350,A 146.128,B 90.000,C 0.000} C_DIS
LIN {X 240.895,Y -161.461,Z 148.308,A 146.168,B 90.000,C 0.000} C_DIS
LIN {X 240.919,Y -161.426,Z 148.257,A 146.176,B 90.000,C 0.000} C_DIS
LIN {X 240.954,Y -161.373,Z 148.206,A 146.189,B 90.000,C 0.000} C_DIS
LIN {X 241.124,Y -161.118,Z 148.163,A 146.249,B 90.000,C 0.000} C_DIS
LIN {X 241.160,Y -161.065,Z 148.112,A 146.262,B 90.000,C 0.000} C_DIS
LIN {X 241.183,Y -161.030,Z 148.061,A 146.270,B 90.000,C 0.000} C_DIS
LIN {X 241.297,Y -160.860,Z 148.019,A 146.311,B 90.000,C 0.000} C_DIS
LIN {X 241.344,Y -160.789,Z 147.917,A 146.327,B 90.000,C 0.000} C_DIS
LIN {X 241.457,Y -160.620,Z 147.874,A 146.368,B 90.000,C 0.000} C_DIS
LIN {X 241.480,Y -160.584,Z 147.823,A 146.376,B 90.000,C 0.000} C_DIS
LIN {X 241.516,Y -160.531,Z 147.772,A 146.389,B 90.000,C 0.000} C_DIS
LIN {X 241.685,Y -160.276,Z 147.730,A 146.449,B 90.000,C 0.000} C_DIS
LIN {X 241.720,Y -160.223,Z 147.679,A 146.462,B 90.000,C 0.000} C_DIS
LIN {X 241.744,Y -160.188,Z 147.628,A 146.470,B 90.000,C 0.000} C_DIS
LIN {X 241.856,Y -160.017,Z 147.585,A 146.511,B 90.000,C 0.000} C_DIS
LIN {X 241.903,Y -159.947,Z 147.483,A 146.527,B 90.000,C 0.000} C_DIS
LIN {X 242.016,Y -159.776,Z 147.441,A 146.568,B 90.000,C 0.000} C_DIS
LIN {X 242.039,Y -159.741,Z 147.390,A 146.576,B 90.000,C 0.000} C_DIS
LIN {X 242.074,Y -159.688,Z 147.339,A 146.589,B 90.000,C 0.000} C_DIS
LIN {X 242.243,Y -159.432,Z 147.296,A 146.649,B 90.000,C 0.000} C_DIS
LIN {X 242.278,Y -159.379,Z 147.245,A 146.662,B 90.000,C 0.000} C_DIS
LIN {X 242.301,Y -159.343,Z 147.194,A 146.670,B 90.000,C 0.000} C_DIS
LIN {X 242.413,Y -159.173,Z 147.152,A 146.710,B 90.000,C 0.000} C_DIS
LIN {X 242.460,Y -159.102,Z 147.050,A 146.727,B 90.000,C 0.000} C_DIS
LIN {X 242.572,Y -158.931,Z 147.007,A 146.767,B 90.000,C 0.000} C_DIS
LIN {X 242.595,Y -158.895,Z 146.956,A 146.776,B 90.000,C 0.000} C_DIS
LIN {X 242.630,Y -158.842,Z 146.905,A 146.788,B 90.000,C 0.000} C_DIS
LIN {X 242.797,Y -158.586,Z 146.863,A 146.849,B 90.000,C 0.000} C_DIS
LIN {X 242.832,Y -158.533,Z 146.812,A 146.862,B 90.000,C 0.000} C_DIS
LIN {X 242.855,Y -158.497,Z 146.761,A 146.870,B 90.000,C 0.000} C_DIS
LIN {X 242.967,Y -158.326,Z 146.718,A 146.910,B 90.000,C 0.000} C_DIS
LIN {X 243.013,Y -158.255,Z 146.616,A 146.927,B 90.000,C 0.000} C_DIS
LIN {X 243.125,Y -158.084,Z 146.574,A 146.967,B 90.000,C 0.000} C_DIS
LIN {X 243.148,Y -158.048,Z 146.522,A 146.976,B 90.000,C 0.000} C_DIS
LIN {X 243.182,Y -157.995,Z 146.471,A 146.988,B 90.000,C 0.000} C_DIS
LIN {X 243.349,Y -157.738,Z 146.429,A 147.049,B 90.000,C 0.000} C_DIS
LIN {X 243.384,Y -157.684,Z 146.378,A 147.061,B 90.000,C 0.000} C_DIS
LIN {X 243.407,Y -157.649,Z 146.327,A 147.070,B 90.000,C 0.000} C_DIS
LIN {X 243.518,Y -157.477,Z 146.284,A 147.110,B 90.000,C 0.000} C_DIS
LIN {X 243.564,Y -157.406,Z 146.182,A 147.127,B 90.000,C 0.000} C_DIS
LIN {X 243.675,Y -157.235,Z 146.140,A 147.167,B 90.000,C 0.000} C_DIS
LIN {X 243.698,Y -157.199,Z 146.089,A 147.176,B 90.000,C 0.000} C_DIS
LIN {X 243.732,Y -157.145,Z 146.038,A 147.188,B 90.000,C 0.000} C_DIS
LIN {X 243.898,Y -156.888,Z 145.995,A 147.249,B 90.000,C 0.000} C_DIS
LIN {X 243.932,Y -156.834,Z 145.944,A 147.261,B 90.000,C 0.000} C_DIS
LIN {X 243.955,Y -156.799,Z 145.893,A 147.270,B 90.000,C 0.000} C_DIS
LIN {X 244.066,Y -156.627,Z 145.851,A 147.310,B 90.000,C 0.000} C_DIS
LIN {X 244.111,Y -156.555,Z 145.749,A 147.327,B 90.000,C 0.000} C_DIS
LIN {X 244.222,Y -156.384,Z 145.706,A 147.367,B 90.000,C 0.000} C_DIS
LIN {X 244.244,Y -156.348,Z 145.655,A 147.376,B 90.000,C 0.000} C_DIS
LIN {X 244.279,Y -156.294,Z 145.604,A 147.388,B 90.000,C 0.000} C_DIS
LIN {X 244.444,Y -156.036,Z 145.562,A 147.449,B 90.000,C 0.000} C_DIS
LIN {X 244.478,Y -155.982,Z 145.511,A 147.461,B 90.000,C 0.000} C_DIS
LIN {X 244.501,Y -155.947,Z 145.460,A 147.470,B 90.000,C 0.000} C_DIS
LIN {X 244.610,Y -155.775,Z 145.417,A 147.510,B 90.000,C 0.000} C_DIS
LIN {X 244.656,Y -155.703,Z 145.315,A 147.527,B 90.000,C 0.000} C_DIS
LIN {X 244.766,Y -155.531,Z 145.273,A 147.567,B 90.000,C 0.000} C_DIS
LIN {X 244.811,Y -155.459,Z 145.171,A 147.584,B 90.000,C 0.000} C_DIS
LIN {X 244.921,Y -155.287,Z 145.128,A 147.624,B 90.000,C 0.000} C_DIS
LIN {X 244.943,Y -155.251,Z 145.077,A 147.633,B 90.000,C 0.000} C_DIS
LIN {X 244.977,Y -155.197,Z 145.026,A 147.645,B 90.000,C 0.000} C_DIS
LIN {X 245.141,Y -154.938,Z 144.984,A 147.706,B 90.000,C 0.000} C_DIS
LIN {X 245.175,Y -154.884,Z 144.933,A 147.718,B 90.000,C 0.000} C_DIS
LIN {X 245.198,Y -154.848,Z 144.882,A 147.727,B 90.000,C 0.000} C_DIS
LIN {X 245.307,Y -154.676,Z 144.839,A 147.767,B 90.000,C 0.000} C_DIS
LIN {X 245.352,Y -154.604,Z 144.737,A 147.784,B 90.000,C 0.000} C_DIS
LIN {X 245.461,Y -154.431,Z 144.695,A 147.824,B 90.000,C 0.000} C_DIS
LIN {X 245.483,Y -154.395,Z 144.644,A 147.832,B 90.000,C 0.000} C_DIS
LIN {X 245.517,Y -154.341,Z 144.593,A 147.845,B 90.000,C 0.000} C_DIS
LIN {X 245.680,Y -154.082,Z 144.550,A 147.905,B 90.000,C 0.000} C_DIS
LIN {X 245.714,Y -154.028,Z 144.499,A 147.918,B 90.000,C 0.000} C_DIS
LIN {X 245.737,Y -153.992,Z 144.448,A 147.926,B 90.000,C 0.000} C_DIS
LIN {X 245.845,Y -153.819,Z 144.406,A 147.967,B 90.000,C 0.000} C_DIS
LIN {X 245.890,Y -153.747,Z 144.304,A 147.984,B 90.000,C 0.000} C_DIS
LIN {X 245.998,Y -153.574,Z 144.261,A 148.024,B 90.000,C 0.000} C_DIS
LIN {X 246.021,Y -153.538,Z 144.210,A 148.032,B 90.000,C 0.000} C_DIS
LIN {X 246.054,Y -153.484,Z 144.159,A 148.045,B 90.000,C 0.000} C_DIS
LIN {X 246.216,Y -153.224,Z 144.117,A 148.105,B 90.000,C 0.000} C_DIS
LIN {X 246.250,Y -153.170,Z 144.066,A 148.118,B 90.000,C 0.000} C_DIS
LIN {X 246.272,Y -153.134,Z 144.014,A 148.126,B 90.000,C 0.000} C_DIS
LIN {X 246.380,Y -152.960,Z 143.972,A 148.167,B 90.000,C 0.000} C_DIS
LIN {X 246.425,Y -152.888,Z 143.870,A 148.183,B 90.000,C 0.000} C_DIS
LIN {X 246.532,Y -152.715,Z 143.828,A 148.224,B 90.000,C 0.000} C_DIS
LIN {X 246.555,Y -152.679,Z 143.776,A 148.232,B 90.000,C 0.000} C_DIS
LIN {X 246.588,Y -152.625,Z 143.725,A 148.245,B 90.000,C 0.000} C_DIS
LIN {X 246.749,Y -152.364,Z 143.683,A 148.305,B 90.000,C 0.000} C_DIS
LIN {X 246.783,Y -152.310,Z 143.632,A 148.318,B 90.000,C 0.000} C_DIS
LIN {X 246.805,Y -152.274,Z 143.581,A 148.326,B 90.000,C 0.000} C_DIS
LIN {X 246.912,Y -152.100,Z 143.538,A 148.367,B 90.000,C 0.000} C_DIS
LIN {X 246.957,Y -152.028,Z 143.436,A 148.383,B 90.000,C 0.000} C_DIS
LIN {X 247.064,Y -151.854,Z 143.394,A 148.424,B 90.000,C 0.000} C_DIS
LIN {X 247.086,Y -151.818,Z 143.343,A 148.432,B 90.000,C 0.000} C_DIS
LIN {X 247.119,Y -151.763,Z 143.292,A 148.445,B 90.000,C 0.000} C_DIS
LIN {X 247.279,Y -151.502,Z 143.249,A 148.505,B 90.000,C 0.000} C_DIS
LIN {X 247.313,Y -151.448,Z 143.198,A 148.518,B 90.000,C 0.000} C_DIS
LIN {X 247.335,Y -151.412,Z 143.147,A 148.526,B 90.000,C 0.000} C_DIS
LIN {X 247.441,Y -151.238,Z 143.105,A 148.566,B 90.000,C 0.000} C_DIS
LIN {X 247.485,Y -151.165,Z 143.003,A 148.583,B 90.000,C 0.000} C_DIS
LIN {X 247.592,Y -150.991,Z 142.960,A 148.624,B 90.000,C 0.000} C_DIS
LIN {X 247.614,Y -150.955,Z 142.909,A 148.632,B 90.000,C 0.000} C_DIS
LIN {X 247.647,Y -150.900,Z 142.858,A 148.645,B 90.000,C 0.000} C_DIS
LIN {X 247.806,Y -150.639,Z 142.816,A 148.705,B 90.000,C 0.000} C_DIS
LIN {X 247.839,Y -150.584,Z 142.765,A 148.718,B 90.000,C 0.000} C_DIS
LIN {X 247.861,Y -150.548,Z 142.714,A 148.726,B 90.000,C 0.000} C_DIS
LIN {X 247.967,Y -150.374,Z 142.671,A 148.766,B 90.000,C 0.000} C_DIS
LIN {X 248.011,Y -150.301,Z 142.569,A 148.783,B 90.000,C 0.000} C_DIS
LIN {X 248.117,Y -150.126,Z 142.527,A 148.823,B 90.000,C 0.000} C_DIS
LIN {X 248.139,Y -150.090,Z 142.476,A 148.832,B 90.000,C 0.000} C_DIS
LIN {X 248.172,Y -150.036,Z 142.425,A 148.844,B 90.000,C 0.000} C_DIS
LIN {X 248.330,Y -149.773,Z 142.382,A 148.905,B 90.000,C 0.000} C_DIS
LIN {X 248.363,Y -149.719,Z 142.331,A 148.917,B 90.000,C 0.000} C_DIS
LIN {X 248.385,Y -149.683,Z 142.280,A 148.926,B 90.000,C 0.000} C_DIS
LIN {X 248.490,Y -149.508,Z 142.238,A 148.966,B 90.000,C 0.000} C_DIS
LIN {X 248.534,Y -149.435,Z 142.136,A 148.983,B 90.000,C 0.000} C_DIS
LIN {X 248.639,Y -149.260,Z 142.093,A 149.023,B 90.000,C 0.000} C_DIS
LIN {X 248.683,Y -149.187,Z 141.991,A 149.040,B 90.000,C 0.000} C_DIS
LIN {X 248.788,Y -149.012,Z 141.949,A 149.080,B 90.000,C 0.000} C_DIS
LIN {X 248.810,Y -148.976,Z 141.898,A 149.089,B 90.000,C 0.000} C_DIS
LIN {X 248.842,Y -148.921,Z 141.847,A 149.101,B 90.000,C 0.000} C_DIS
LIN {X 249.000,Y -148.658,Z 141.804,A 149.162,B 90.000,C 0.000} C_DIS
LIN {X 249.032,Y -148.603,Z 141.753,A 149.174,B 90.000,C 0.000} C_DIS
LIN {X 249.054,Y -148.567,Z 141.702,A 149.183,B 90.000,C 0.000} C_DIS
LIN {X 249.158,Y -148.392,Z 141.660,A 149.223,B 90.000,C 0.000} C_DIS
LIN {X 249.202,Y -148.319,Z 141.558,A 149.240,B 90.000,C 0.000} C_DIS
LIN {X 249.306,Y -148.143,Z 141.515,A 149.280,B 90.000,C 0.000} C_DIS
LIN {X 249.328,Y -148.107,Z 141.464,A 149.289,B 90.000,C 0.000} C_DIS
LIN {X 249.360,Y -148.052,Z 141.413,A 149.301,B 90.000,C 0.000} C_DIS
LIN {X 249.517,Y -147.788,Z 141.371,A 149.362,B 90.000,C 0.000} C_DIS
LIN {X 249.549,Y -147.734,Z 141.319,A 149.374,B 90.000,C 0.000} C_DIS
LIN {X 249.571,Y -147.697,Z 141.268,A 149.383,B 90.000,C 0.000} C_DIS
LIN {X 249.675,Y -147.521,Z 141.226,A 149.423,B 90.000,C 0.000} C_DIS
LIN {X 249.718,Y -147.448,Z 141.124,A 149.440,B 90.000,C 0.000} C_DIS
LIN {X 249.822,Y -147.272,Z 141.081,A 149.480,B 90.000,C 0.000} C_DIS
LIN {X 249.843,Y -147.236,Z 141.030,A 149.489,B 90.000,C 0.000} C_DIS
LIN {X 249.875,Y -147.181,Z 140.979,A 149.501,B 90.000,C 0.000} C_DIS
LIN {X 250.031,Y -146.917,Z 140.937,A 149.562,B 90.000,C 0.000} C_DIS
LIN {X 250.063,Y -146.862,Z 140.886,A 149.574,B 90.000,C 0.000} C_DIS
LIN {X 250.084,Y -146.826,Z 140.835,A 149.583,B 90.000,C 0.000} C_DIS
LIN {X 250.188,Y -146.650,Z 140.792,A 149.623,B 90.000,C 0.000} C_DIS
LIN {X 250.231,Y -146.576,Z 140.690,A 149.640,B 90.000,C 0.000} C_DIS
LIN {X 250.334,Y -146.400,Z 140.648,A 149.680,B 90.000,C 0.000} C_DIS
LIN {X 250.355,Y -146.363,Z 140.597,A 149.688,B 90.000,C 0.000} C_DIS
LIN {X 250.387,Y -146.308,Z 140.546,A 149.701,B 90.000,C 0.000} C_DIS
LIN {X 250.542,Y -146.044,Z 140.503,A 149.762,B 90.000,C 0.000} C_DIS
LIN {X 250.574,Y -145.989,Z 140.452,A 149.774,B 90.000,C 0.000} C_DIS
LIN {X 250.590,Y -145.961,Z 140.401,A 149.781,B 90.000,C 0.000} C_DIS
LIN {X 250.630,Y -145.892,Z 140.380,A 149.796,B 90.000,C 0.000} C_DIS
LIN {X 250.696,Y -145.779,Z 140.328,A 149.822,B 90.000,C 0.000} C_DIS
LIN {X 250.775,Y -145.643,Z 140.203,A 149.853,B 90.000,C 0.000} C_DIS
LIN {X 250.847,Y -145.519,Z 139.982,A 149.882,B 90.000,C 0.000} C_DIS
LIN {X 250.875,Y -145.471,Z 139.342,A 149.893,B 90.000,C 0.000} C_DIS
LIN {X 250.926,Y -145.382,Z 139.118,A 149.913,B 90.000,C 0.000} C_DIS
LIN {X 250.937,Y -145.364,Z 138.863,A 149.917,B 90.000,C 0.000} C_DIS
LIN {X 250.922,Y -145.389,Z 138.549,A 149.911,B 90.000,C 0.000} C_DIS
LIN {X 250.890,Y -145.445,Z 138.508,A 149.898,B 90.000,C 0.000} C_DIS
LIN {X 250.751,Y -145.684,Z 138.480,A 149.844,B 90.000,C 0.000} C_DIS
LIN {X 250.719,Y -145.739,Z 138.429,A 149.831,B 90.000,C 0.000} C_DIS
LIN {X 250.698,Y -145.776,Z 138.378,A 149.823,B 90.000,C 0.000} C_DIS
LIN {X 250.595,Y -145.952,Z 138.335,A 149.783,B 90.000,C 0.000} C_DIS
LIN {X 250.574,Y -145.989,Z 138.284,A 149.774,B 90.000,C 0.000} C_DIS
LIN {X 250.542,Y -146.044,Z 138.233,A 149.762,B 90.000,C 0.000} C_DIS
LIN {X 250.387,Y -146.308,Z 138.191,A 149.701,B 90.000,C 0.000} C_DIS
LIN {X 250.355,Y -146.363,Z 138.140,A 149.688,B 90.000,C 0.000} C_DIS
LIN {X 250.334,Y -146.400,Z 138.089,A 149.680,B 90.000,C 0.000} C_DIS
LIN {X 250.231,Y -146.576,Z 138.046,A 149.640,B 90.000,C 0.000} C_DIS
LIN {X 250.188,Y -146.650,Z 137.944,A 149.623,B 90.000,C 0.000} C_DIS
LIN {X 250.084,Y -146.826,Z 137.902,A 149.583,B 90.000,C 0.000} C_DIS
LIN {X 250.063,Y -146.862,Z 137.851,A 149.574,B 90.000,C 0.000} C_DIS
LIN {X 250.031,Y -146.917,Z 137.800,A 149.562,B 90.000,C 0.000} C_DIS
LIN {X 249.875,Y -147.181,Z 137.757,A 149.501,B 90.000,C 0.000} C_DIS
LIN {X 249.843,Y -147.236,Z 137.706,A 149.489,B 90.000,C 0.000} C_DIS
LIN {X 249.822,Y -147.272,Z 137.655,A 149.480,B 90.000,C 0.000} C_DIS
LIN {X 249.718,Y -147.448,Z 137.613,A 149.440,B 90.000,C 0.000} C_DIS
LIN {X 249.675,Y -147.521,Z 137.511,A 149.423,B 90.000,C 0.000} C_DIS
LIN {X 249.571,Y -147.697,Z 137.468,A 149.383,B 90.000,C 0.000} C_DIS
LIN {X 249.549,Y -147.734,Z 137.417,A 149.374,B 90.000,C 0.000} C_DIS
LIN {X 249.517,Y -147.788,Z 137.366,A 149.362,B 90.000,C 0.000} C_DIS
LIN {X 249.360,Y -148.052,Z 137.324,A 149.301,B 90.000,C 0.000} C_DIS
LIN {X 249.328,Y -148.107,Z 137.273,A 149.289,B 90.000,C 0.000} C_DIS
LIN {X 249.306,Y -148.143,Z 137.222,A 149.280,B 90.000,C 0.000} C_DIS
LIN {X 249.202,Y -148.319,Z 137.179,A 149.240,B 90.000,C 0.000} C_DIS
LIN {X 249.180,Y -148.355,Z 137.128,A 149.232,B 90.000,C 0.000} C_DIS
LIN {X 249.148,Y -148.410,Z 137.077,A 149.219,B 90.000,C 0.000} C_DIS
LIN {X 248.991,Y -148.673,Z 137.035,A 149.159,B 90.000,C 0.000} C_DIS
LIN {X 248.958,Y -148.727,Z 136.984,A 149.146,B 90.000,C 0.000} C_DIS
LIN {X 248.936,Y -148.764,Z 136.933,A 149.138,B 90.000,C 0.000} C_DIS
LIN {X 248.832,Y -148.939,Z 136.890,A 149.097,B 90.000,C 0.000} C_DIS
LIN {X 248.788,Y -149.012,Z 136.788,A 149.080,B 90.000,C 0.000} C_DIS
LIN {X 248.683,Y -149.187,Z 136.746,A 149.040,B 90.000,C 0.000} C_DIS
LIN {X 248.661,Y -149.223,Z 136.695,A 149.032,B 90.000,C 0.000} C_DIS
LIN {X 248.628,Y -149.278,Z 136.644,A 149.019,B 90.000,C 0.000} C_DIS
LIN {X 248.471,Y -149.541,Z 136.601,A 148.959,B 90.000,C 0.000} C_DIS
LIN {X 248.438,Y -149.595,Z 136.550,A 148.946,B 90.000,C 0.000} C_DIS
LIN {X 248.416,Y -149.631,Z 136.499,A 148.938,B 90.000,C 0.000} C_DIS
LIN {X 248.310,Y -149.806,Z 136.457,A 148.897,B 90.000,C 0.000} C_DIS
LIN {X 248.289,Y -149.843,Z 136.406,A 148.889,B 90.000,C 0.000} C_DIS
LIN {X 248.256,Y -149.897,Z 136.354,A 148.876,B 90.000,C 0.000} C_DIS
LIN {X 248.097,Y -150.159,Z 136.312,A 148.816,B 90.000,C 0.000} C_DIS
LIN {X 248.064,Y -150.214,Z 136.261,A 148.803,B 90.000,C 0.000} C_DIS
LIN {X 248.042,Y -150.250,Z 136.210,A 148.795,B 90.000,C 0.000} C_DIS
LIN {X 247.936,Y -150.425,Z 136.168,A 148.755,B 90.000,C 0.000} C_DIS
LIN {X 247.892,Y -150.497,Z 136.065,A 148.738,B 90.000,C 0.000} C_DIS
LIN {X 247.786,Y -150.672,Z 136.023,A 148.697,B 90.000,C 0.000} C_DIS
LIN {X 247.764,Y -150.708,Z 135.972,A 148.689,B 90.000,C 0.000} C_DIS
LIN {X 247.731,Y -150.762,Z 135.921,A 148.676,B 90.000,C 0.000} C_DIS
LIN {X 247.572,Y -151.024,Z 135.878,A 148.616,B 90.000,C 0.000} C_DIS
LIN {X 247.539,Y -151.078,Z 135.827,A 148.603,B 90.000,C 0.000} C_DIS
LIN {X 247.517,Y -151.114,Z 135.776,A 148.595,B 90.000,C 0.000} C_DIS
LIN {X 247.410,Y -151.289,Z 135.734,A 148.555,B 90.000,C 0.000} C_DIS
LIN {X 247.366,Y -151.361,Z 135.632,A 148.538,B 90.000,C 0.000} C_DIS
LIN {X 247.259,Y -151.535,Z 135.589,A 148.498,B 90.000,C 0.000} C_DIS
LIN {X 247.237,Y -151.571,Z 135.538,A 148.489,B 90.000,C 0.000} C_DIS
LIN {X 247.204,Y -151.626,Z 135.487,A 148.477,B 90.000,C 0.000} C_DIS
LIN {X 247.043,Y -151.887,Z 135.445,A 148.416,B 90.000,C 0.000} C_DIS
LIN {X 247.010,Y -151.941,Z 135.394,A 148.404,B 90.000,C 0.000} C_DIS
LIN {X 246.988,Y -151.977,Z 135.343,A 148.395,B 90.000,C 0.000} C_DIS
LIN {X 246.881,Y -152.151,Z 135.300,A 148.355,B 90.000,C 0.000} C_DIS
LIN {X 246.859,Y -152.187,Z 135.249,A 148.346,B 90.000,C 0.000} C_DIS
LIN {X 246.825,Y -152.241,Z 135.198,A 148.334,B 90.000,C 0.000} C_DIS
LIN {X 246.664,Y -152.502,Z 135.156,A 148.273,B 90.000,C 0.000} C_DIS
LIN {X 246.631,Y -152.556,Z 135.105,A 148.261,B 90.000,C 0.000} C_DIS
LIN {X 246.608,Y -152.592,Z 135.054,A 148.252,B 90.000,C 0.000} C_DIS
LIN {X 246.501,Y -152.766,Z 135.011,A 148.212,B 90.000,C 0.000} C_DIS
LIN {X 246.456,Y -152.838,Z 134.909,A 148.195,B 90.000,C 0.000} C_DIS
LIN {X 246.349,Y -153.011,Z 134.867,A 148.155,B 90.000,C 0.000} C_DIS
LIN {X 246.326,Y -153.047,Z 134.816,A 148.147,B 90.000,C 0.000} C_DIS
LIN {X 246.292,Y -153.101,Z 134.765,A 148.134,B 90.000,C 0.000} C_DIS
LIN {X 246.131,Y -153.361,Z 134.722,A 148.073,B 90.000,C 0.000} C_DIS
LIN {X 246.097,Y -153.415,Z 134.671,A 148.061,B 90.000,C 0.000} C_DIS
LIN {X 246.075,Y -153.451,Z 134.620,A 148.052,B 90.000,C 0.000} C_DIS
LIN {X 245.966,Y -153.625,Z 134.578,A 148.012,B 90.000,C 0.000} C_DIS
LIN {X 245.944,Y -153.661,Z 134.527,A 148.004,B 90.000,C 0.000} C_DIS
LIN {X 245.910,Y -153.715,Z 134.476,A 147.991,B 90.000,C 0.000} C_DIS
LIN {X 245.748,Y -153.974,Z 134.433,A 147.931,B 90.000,C 0.000} C_DIS
LIN {X 245.714,Y -154.028,Z 134.382,A 147.918,B 90.000,C 0.000} C_DIS
LIN {X 245.691,Y -154.064,Z 134.331,A 147.910,B 90.000,C 0.000} C_DIS
LIN {X 245.583,Y -154.237,Z 134.289,A 147.869,B 90.000,C 0.000} C_DIS
LIN {X 245.538,Y -154.309,Z 134.187,A 147.853,B 90.000,C 0.000} C_DIS
LIN {X 245.429,Y -154.482,Z 134.144,A 147.812,B 90.000,C 0.000} C_DIS
LIN {X 245.406,Y -154.518,Z 134.093,A 147.804,B 90.000,C 0.000} C_DIS
LIN {X 245.372,Y -154.571,Z 134.042,A 147.791,B 90.000,C 0.000} C_DIS
LIN {X 245.209,Y -154.831,Z 134.000,A 147.731,B 90.000,C 0.000} C_DIS
LIN {X 245.175,Y -154.884,Z 133.949,A 147.718,B 90.000,C 0.000} C_DIS
LIN {X 245.152,Y -154.920,Z 133.898,A 147.710,B 90.000,C 0.000} C_DIS
LIN {X 245.043,Y -155.093,Z 133.855,A 147.669,B 90.000,C 0.000} C_DIS
LIN {X 245.021,Y -155.129,Z 133.804,A 147.661,B 90.000,C 0.000} C_DIS
LIN {X 244.987,Y -155.182,Z 133.753,A 147.648,B 90.000,C 0.000} C_DIS
LIN {X 244.823,Y -155.441,Z 133.711,A 147.588,B 90.000,C 0.000} C_DIS
LIN {X 244.788,Y -155.495,Z 133.659,A 147.575,B 90.000,C 0.000} C_DIS
LIN {X 244.766,Y -155.531,Z 133.608,A 147.567,B 90.000,C 0.000} C_DIS
LIN {X 244.656,Y -155.703,Z 133.566,A 147.527,B 90.000,C 0.000} C_DIS
LIN {X 244.610,Y -155.775,Z 133.464,A 147.510,B 90.000,C 0.000} C_DIS
LIN {X 244.501,Y -155.947,Z 133.421,A 147.470,B 90.000,C 0.000} C_DIS
LIN {X 244.478,Y -155.982,Z 133.370,A 147.461,B 90.000,C 0.000} C_DIS
LIN {X 244.444,Y -156.036,Z 133.319,A 147.449,B 90.000,C 0.000} C_DIS
LIN {X 244.279,Y -156.294,Z 133.277,A 147.388,B 90.000,C 0.000} C_DIS
LIN {X 244.244,Y -156.348,Z 133.226,A 147.376,B 90.000,C 0.000} C_DIS
LIN {X 244.222,Y -156.384,Z 133.175,A 147.367,B 90.000,C 0.000} C_DIS
LIN {X 244.111,Y -156.555,Z 133.132,A 147.327,B 90.000,C 0.000} C_DIS
LIN {X 244.066,Y -156.627,Z 133.030,A 147.310,B 90.000,C 0.000} C_DIS
LIN {X 243.955,Y -156.799,Z 132.988,A 147.270,B 90.000,C 0.000} C_DIS
LIN {X 243.932,Y -156.834,Z 132.937,A 147.261,B 90.000,C 0.000} C_DIS
LIN {X 243.898,Y -156.888,Z 132.886,A 147.249,B 90.000,C 0.000} C_DIS
LIN {X 243.732,Y -157.145,Z 132.843,A 147.188,B 90.000,C 0.000} C_DIS
LIN {X 243.698,Y -157.199,Z 132.792,A 147.176,B 90.000,C 0.000} C_DIS
LIN {X 243.675,Y -157.235,Z 132.741,A 147.167,B 90.000,C 0.000} C_DIS
LIN {X 243.564,Y -157.406,Z 132.699,A 147.127,B 90.000,C 0.000} C_DIS
LIN {X 243.541,Y -157.442,Z 132.648,A 147.119,B 90.000,C 0.000} C_DIS
LIN {X 243.506,Y -157.495,Z 132.597,A 147.106,B 90.000,C 0.000} C_DIS
LIN {X 243.340,Y -157.752,Z 132.554,A 147.045,B 90.000,C 0.000} C_DIS
LIN {X 243.305,Y -157.806,Z 132.503,A 147.033,B 90.000,C 0.000} C_DIS
LIN {X 243.282,Y -157.841,Z 132.452,A 147.024,B 90.000,C 0.000} C_DIS
LIN {X 243.171,Y -158.013,Z 132.410,A 146.984,B 90.000,C 0.000} C_DIS
LIN {X 243.125,Y -158.084,Z 132.308,A 146.967,B 90.000,C 0.000} C_DIS
LIN {X 243.013,Y -158.255,Z 132.265,A 146.927,B 90.000,C 0.000} C_DIS
LIN {X 242.990,Y -158.290,Z 132.214,A 146.919,B 90.000,C 0.000} C_DIS
LIN {X 242.955,Y -158.344,Z 132.163,A 146.906,B 90.000,C 0.000} C_DIS
LIN {X 242.788,Y -158.600,Z 132.121,A 146.846,B 90.000,C 0.000} C_DIS
LIN {X 242.753,Y -158.654,Z 132.070,A 146.833,B 90.000,C 0.000} C_DIS
LIN {X 242.730,Y -158.689,Z 132.019,A 146.825,B 90.000,C 0.000} C_DIS
LIN {X 242.618,Y -158.860,Z 131.976,A 146.784,B 90.000,C 0.000} C_DIS
LIN {X 242.595,Y -158.895,Z 131.925,A 146.776,B 90.000,C 0.000} C_DIS
LIN {X 242.560,Y -158.949,Z 131.874,A 146.763,B 90.000,C 0.000} C_DIS
LIN {X 242.392,Y -159.205,Z 131.832,A 146.703,B 90.000,C 0.000} C_DIS
LIN {X 242.357,Y -159.258,Z 131.781,A 146.690,B 90.000,C 0.000} C_DIS
LIN {X 242.334,Y -159.293,Z 131.730,A 146.682,B 90.000,C 0.000} C_DIS
LIN {X 242.221,Y -159.464,Z 131.687,A 146.642,B 90.000,C 0.000} C_DIS
LIN {X 242.175,Y -159.535,Z 131.585,A 146.625,B 90.000,C 0.000} C_DIS
LIN {X 242.062,Y -159.705,Z 131.543,A 146.584,B 90.000,C 0.000} C_DIS
LIN {X 242.039,Y -159.741,Z 131.492,A 146.576,B 90.000,C 0.000} C_DIS
LIN {X 242.004,Y -159.794,Z 131.441,A 146.563,B 90.000,C 0.000} C_DIS
LIN {X 241.835,Y -160.049,Z 131.398,A 146.503,B 90.000,C 0.000} C_DIS
LIN {X 241.800,Y -160.102,Z 131.347,A 146.490,B 90.000,C 0.000} C_DIS
LIN {X 241.776,Y -160.138,Z 131.296,A 146.482,B 90.000,C 0.000} C_DIS
LIN {X 241.664,Y -160.308,Z 131.254,A 146.442,B 90.000,C 0.000} C_DIS
LIN {X 241.640,Y -160.343,Z 131.203,A 146.433,B 90.000,C 0.000} C_DIS
LIN {X 241.605,Y -160.396,Z 131.151,A 146.421,B 90.000,C 0.000} C_DIS
LIN {X 241.435,Y -160.652,Z 131.109,A 146.360,B 90.000,C 0.000} C_DIS
LIN {X 241.400,Y -160.705,Z 131.058,A 146.348,B 90.000,C 0.000} C_DIS
LIN {X 241.377,Y -160.740,Z 131.007,A 146.339,B 90.000,C 0.000} C_DIS
LIN {X 241.263,Y -160.910,Z 130.964,A 146.299,B 90.000,C 0.000} C_DIS
LIN {X 241.216,Y -160.980,Z 130.862,A 146.282,B 90.000,C 0.000} C_DIS
LIN {X 241.103,Y -161.150,Z 130.820,A 146.242,B 90.000,C 0.000} C_DIS
LIN {X 241.079,Y -161.185,Z 130.769,A 146.233,B 90.000,C 0.000} C_DIS
LIN {X 241.044,Y -161.238,Z 130.718,A 146.221,B 90.000,C 0.000} C_DIS
LIN {X 240.874,Y -161.493,Z 130.675,A 146.160,B 90.000,C 0.000} C_DIS
LIN {X 240.838,Y -161.546,Z 130.624,A 146.148,B 90.000,C 0.000} C_DIS
LIN {X 240.814,Y -161.581,Z 130.573,A 146.139,B 90.000,C 0.000} C_DIS
LIN {X 240.701,Y -161.750,Z 130.531,A 146.099,B 90.000,C 0.000} C_DIS
LIN {X 240.653,Y -161.821,Z 130.429,A 146.082,B 90.000,C 0.000} C_DIS
LIN {X 240.539,Y -161.990,Z 130.386,A 146.042,B 90.000,C 0.000} C_DIS
LIN {X 240.516,Y -162.025,Z 130.335,A 146.033,B 90.000,C 0.000} C_DIS
LIN {X 240.480,Y -162.078,Z 130.284,A 146.021,B 90.000,C 0.000} C_DIS
LIN {X 240.309,Y -162.332,Z 130.242,A 145.960,B 90.000,C 0.000} C_DIS
LIN {X 240.273,Y -162.385,Z 130.191,A 145.948,B 90.000,C 0.000} C_DIS
LIN {X 240.249,Y -162.420,Z 130.140,A 145.939,B 90.000,C 0.000} C_DIS
LIN {X 240.135,Y -162.589,Z 130.097,A 145.899,B 90.000,C 0.000} C_DIS
LIN {X 240.111,Y -162.624,Z 130.046,A 145.891,B 90.000,C 0.000} C_DIS
LIN {X 240.075,Y -162.677,Z 129.995,A 145.878,B 90.000,C 0.000} C_DIS
LIN {X 239.903,Y -162.930,Z 129.953,A 145.818,B 90.000,C 0.000} C_DIS
LIN {X 239.868,Y -162.983,Z 129.902,A 145.805,B 90.000,C 0.000} C_DIS
LIN {X 239.844,Y -163.018,Z 129.851,A 145.797,B 90.000,C 0.000} C_DIS
LIN {X 239.729,Y -163.187,Z 129.808,A 145.756,B 90.000,C 0.000} C_DIS
LIN {X 239.681,Y -163.257,Z 129.706,A 145.740,B 90.000,C 0.000} C_DIS
LIN {X 239.566,Y -163.426,Z 129.664,A 145.699,B 90.000,C 0.000} C_DIS
LIN {X 239.542,Y -163.461,Z 129.613,A 145.691,B 90.000,C 0.000} C_DIS
LIN {X 239.506,Y -163.514,Z 129.562,A 145.678,B 90.000,C 0.000} C_DIS
LIN {X 239.334,Y -163.766,Z 129.519,A 145.618,B 90.000,C 0.000} C_DIS
LIN {X 239.298,Y -163.819,Z 129.468,A 145.605,B 90.000,C 0.000} C_DIS
LIN {X 239.274,Y -163.854,Z 129.417,A 145.597,B 90.000,C 0.000} C_DIS
LIN {X 239.158,Y -164.022,Z 129.375,A 145.556,B 90.000,C 0.000} C_DIS
LIN {X 239.134,Y -164.057,Z 129.324,A 145.548,B 90.000,C 0.000} C_DIS
LIN {X 239.098,Y -164.110,Z 129.273,A 145.535,B 90.000,C 0.000} C_DIS
LIN {X 238.925,Y -164.362,Z 129.230,A 145.475,B 90.000,C 0.000} C_DIS
LIN {X 238.889,Y -164.415,Z 129.179,A 145.462,B 90.000,C 0.000} C_DIS
LIN {X 238.865,Y -164.450,Z 129.128,A 145.454,B 90.000,C 0.000} C_DIS
LIN {X 238.749,Y -164.618,Z 129.086,A 145.414,B 90.000,C 0.000} C_DIS
LIN {X 238.701,Y -164.688,Z 128.984,A 145.397,B 90.000,C 0.000} C_DIS
LIN {X 238.585,Y -164.856,Z 128.941,A 145.357,B 90.000,C 0.000} C_DIS
LIN {X 238.560,Y -164.891,Z 128.890,A 145.348,B 90.000,C 0.000} C_DIS
LIN {X 238.524,Y -164.943,Z 128.839,A 145.336,B 90.000,C 0.000} C_DIS
LIN {X 238.350,Y -165.195,Z 128.797,A 145.275,B 90.000,C 0.000} C_DIS
LIN {X 238.314,Y -165.247,Z 128.746,A 145.262,B 90.000,C 0.000} C_DIS
LIN {X 238.289,Y -165.282,Z 128.695,A 145.254,B 90.000,C 0.000} C_DIS
LIN {X 238.173,Y -165.450,Z 128.652,A 145.214,B 90.000,C 0.000} C_DIS
LIN {X 238.149,Y -165.485,Z 128.601,A 145.205,B 90.000,C 0.000} C_DIS
LIN {X 238.112,Y -165.537,Z 128.550,A 145.193,B 90.000,C 0.000} C_DIS
LIN {X 237.938,Y -165.788,Z 128.508,A 145.132,B 90.000,C 0.000} C_DIS
LIN {X 237.901,Y -165.840,Z 128.456,A 145.120,B 90.000,C 0.000} C_DIS
LIN {X 237.877,Y -165.875,Z 128.405,A 145.111,B 90.000,C 0.000} C_DIS
LIN {X 237.760,Y -166.043,Z 128.363,A 145.071,B 90.000,C 0.000} C_DIS
LIN {X 237.711,Y -166.112,Z 128.261,A 145.054,B 90.000,C 0.000} C_DIS
LIN {X 237.594,Y -166.280,Z 128.218,A 145.014,B 90.000,C 0.000} C_DIS
LIN {X 237.570,Y -166.314,Z 128.167,A 145.005,B 90.000,C 0.000} C_DIS
LIN {X 237.534,Y -166.367,Z 128.116,A 144.993,B 90.000,C 0.000} C_DIS
LIN {X 237.358,Y -166.617,Z 128.074,A 144.932,B 90.000,C 0.000} C_DIS
LIN {X 237.321,Y -166.669,Z 128.023,A 144.920,B 90.000,C 0.000} C_DIS
LIN {X 237.297,Y -166.704,Z 127.972,A 144.911,B 90.000,C 0.000} C_DIS
LIN {X 237.179,Y -166.871,Z 127.929,A 144.871,B 90.000,C 0.000} C_DIS
LIN {X 237.130,Y -166.941,Z 127.827,A 144.854,B 90.000,C 0.000} C_DIS
LIN {X 237.013,Y -167.107,Z 127.785,A 144.814,B 90.000,C 0.000} C_DIS
LIN {X 236.988,Y -167.142,Z 127.734,A 144.806,B 90.000,C 0.000} C_DIS
LIN {X 236.952,Y -167.194,Z 127.683,A 144.793,B 90.000,C 0.000} C_DIS
LIN {X 236.775,Y -167.444,Z 127.640,A 144.733,B 90.000,C 0.000} C_DIS
LIN {X 236.738,Y -167.496,Z 127.589,A 144.720,B 90.000,C 0.000} C_DIS
LIN {X 236.714,Y -167.531,Z 127.538,A 144.712,B 90.000,C 0.000} C_DIS
LIN {X 236.596,Y -167.698,Z 127.496,A 144.671,B 90.000,C 0.000} C_DIS
LIN {X 236.571,Y -167.732,Z 127.445,A 144.663,B 90.000,C 0.000} C_DIS
LIN {X 236.534,Y -167.784,Z 127.394,A 144.650,B 90.000,C 0.000} C_DIS
LIN {X 236.357,Y -168.034,Z 127.351,A 144.590,B 90.000,C 0.000} C_DIS
LIN {X 236.320,Y -168.086,Z 127.300,A 144.577,B 90.000,C 0.000} C_DIS
LIN {X 236.296,Y -168.120,Z 127.249,A 144.569,B 90.000,C 0.000} C_DIS
LIN {X 236.177,Y -168.287,Z 127.207,A 144.528,B 90.000,C 0.000} C_DIS
LIN {X 236.128,Y -168.356,Z 127.105,A 144.512,B 90.000,C 0.000} C_DIS
LIN {X 236.009,Y -168.522,Z 127.062,A 144.471,B 90.000,C 0.000} C_DIS
LIN {X 235.985,Y -168.556,Z 127.011,A 144.463,B 90.000,C 0.000} C_DIS
LIN {X 235.948,Y -168.608,Z 126.960,A 144.450,B 90.000,C 0.000} C_DIS
LIN {X 235.769,Y -168.857,Z 126.918,A 144.390,B 90.000,C 0.000} C_DIS
LIN {X 235.732,Y -168.909,Z 126.867,A 144.377,B 90.000,C 0.000} C_DIS
LIN {X 235.708,Y -168.944,Z 126.816,A 144.369,B 90.000,C 0.000} C_DIS
LIN {X 235.589,Y -169.109,Z 126.773,A 144.329,B 90.000,C 0.000} C_DIS
LIN {X 235.564,Y -169.144,Z 126.722,A 144.320,B 90.000,C 0.000} C_DIS
LIN {X 235.527,Y -169.196,Z 126.671,A 144.308,B 90.000,C 0.000} C_DIS
LIN {X 235.348,Y -169.444,Z 126.629,A 144.247,B 90.000,C 0.000} C_DIS
LIN {X 235.311,Y -169.496,Z 126.578,A 144.235,B 90.000,C 0.000} C_DIS
LIN {X 235.286,Y -169.530,Z 126.527,A 144.226,B 90.000,C 0.000} C_DIS
LIN {X 235.166,Y -169.696,Z 126.484,A 144.186,B 90.000,C 0.000} C_DIS
LIN {X 235.117,Y -169.765,Z 126.382,A 144.169,B 90.000,C 0.000} C_DIS
LIN {X 234.997,Y -169.930,Z 126.340,A 144.129,B 90.000,C 0.000} C_DIS
LIN {X 234.972,Y -169.965,Z 126.289,A 144.120,B 90.000,C 0.000} C_DIS
LIN {X 234.935,Y -170.016,Z 126.238,A 144.108,B 90.000,C 0.000} C_DIS
LIN {X 234.755,Y -170.264,Z 126.195,A 144.047,B 90.000,C 0.000} C_DIS
LIN {X 234.718,Y -170.316,Z 126.144,A 144.035,B 90.000,C 0.000} C_DIS
LIN {X 234.693,Y -170.350,Z 126.093,A 144.026,B 90.000,C 0.000} C_DIS
LIN {X 234.573,Y -170.515,Z 126.051,A 143.986,B 90.000,C 0.000} C_DIS
LIN {X 234.548,Y -170.550,Z 125.999,A 143.978,B 90.000,C 0.000} C_DIS
LIN {X 234.511,Y -170.601,Z 125.948,A 143.965,B 90.000,C 0.000} C_DIS
LIN {X 234.330,Y -170.849,Z 125.906,A 143.904,B 90.000,C 0.000} C_DIS
LIN {X 234.293,Y -170.900,Z 125.855,A 143.892,B 90.000,C 0.000} C_DIS
LIN {X 234.268,Y -170.935,Z 125.804,A 143.883,B 90.000,C 0.000} C_DIS
LIN {X 234.147,Y -171.099,Z 125.761,A 143.843,B 90.000,C 0.000} C_DIS
LIN {X 234.097,Y -171.168,Z 125.659,A 143.826,B 90.000,C 0.000} C_DIS
LIN {X 233.977,Y -171.333,Z 125.617,A 143.786,B 90.000,C 0.000} C_DIS
LIN {X 233.952,Y -171.367,Z 125.566,A 143.778,B 90.000,C 0.000} C_DIS
LIN {X 233.914,Y -171.418,Z 125.515,A 143.765,B 90.000,C 0.000} C_DIS
LIN {X 233.733,Y -171.665,Z 125.472,A 143.705,B 90.000,C 0.000} C_DIS
LIN {X 233.695,Y -171.717,Z 125.421,A 143.692,B 90.000,C 0.000} C_DIS
LIN {X 233.670,Y -171.751,Z 125.370,A 143.684,B 90.000,C 0.000} C_DIS
LIN {X 233.549,Y -171.915,Z 125.328,A 143.643,B 90.000,C 0.000} C_DIS
LIN {X 233.499,Y -171.984,Z 125.226,A 143.626,B 90.000,C 0.000} C_DIS
LIN {X 233.378,Y -172.148,Z 125.183,A 143.586,B 90.000,C 0.000} C_DIS
LIN {X 233.352,Y -172.182,Z 125.132,A 143.578,B 90.000,C 0.000} C_DIS
LIN {X 233.315,Y -172.233,Z 125.081,A 143.565,B 90.000,C 0.000} C_DIS
LIN {X 233.133,Y -172.480,Z 125.039,A 143.505,B 90.000,C 0.000} C_DIS
LIN {X 233.095,Y -172.531,Z 124.988,A 143.492,B 90.000,C 0.000} C_DIS
LIN {X 233.069,Y -172.565,Z 124.937,A 143.484,B 90.000,C 0.000} C_DIS
LIN {X 232.948,Y -172.729,Z 124.894,A 143.443,B 90.000,C 0.000} C_DIS
LIN {X 232.923,Y -172.763,Z 124.843,A 143.435,B 90.000,C 0.000} C_DIS
LIN {X 232.885,Y -172.814,Z 124.792,A 143.422,B 90.000,C 0.000} C_DIS
LIN {X 232.702,Y -173.060,Z 124.750,A 143.362,B 90.000,C 0.000} C_DIS
LIN {X 232.664,Y -173.111,Z 124.699,A 143.349,B 90.000,C 0.000} C_DIS
LIN {X 232.639,Y -173.145,Z 124.648,A 143.341,B 90.000,C 0.000} C_DIS
LIN {X 232.517,Y -173.309,Z 124.605,A 143.301,B 90.000,C 0.000} C_DIS
LIN {X 232.466,Y -173.377,Z 124.503,A 143.284,B 90.000,C 0.000} C_DIS
LIN {X 232.344,Y -173.541,Z 124.461,A 143.243,B 90.000,C 0.000} C_DIS
LIN {X 232.318,Y -173.575,Z 124.410,A 143.235,B 90.000,C 0.000} C_DIS
LIN {X 232.280,Y -173.626,Z 124.359,A 143.223,B 90.000,C 0.000} C_DIS
LIN {X 232.097,Y -173.871,Z 124.316,A 143.162,B 90.000,C 0.000} C_DIS
LIN {X 232.059,Y -173.922,Z 124.265,A 143.149,B 90.000,C 0.000} C_DIS
LIN {X 232.033,Y -173.956,Z 124.214,A 143.141,B 90.000,C 0.000} C_DIS
LIN {X 231.911,Y -174.119,Z 124.172,A 143.101,B 90.000,C 0.000} C_DIS
LIN {X 231.885,Y -174.153,Z 124.121,A 143.092,B 90.000,C 0.000} C_DIS
LIN {X 231.847,Y -174.204,Z 124.070,A 143.080,B 90.000,C 0.000} C_DIS
LIN {X 231.663,Y -174.449,Z 124.027,A 143.019,B 90.000,C 0.000} C_DIS
LIN {X 231.625,Y -174.499,Z 123.976,A 143.007,B 90.000,C 0.000} C_DIS
LIN {X 231.599,Y -174.533,Z 123.925,A 142.998,B 90.000,C 0.000} C_DIS
LIN {X 231.476,Y -174.696,Z 123.883,A 142.958,B 90.000,C 0.000} C_DIS
LIN {X 231.425,Y -174.764,Z 123.781,A 142.941,B 90.000,C 0.000} C_DIS
LIN {X 231.302,Y -174.927,Z 123.738,A 142.901,B 90.000,C 0.000} C_DIS
LIN {X 231.276,Y -174.961,Z 123.687,A 142.892,B 90.000,C 0.000} C_DIS
LIN {X 231.238,Y -175.012,Z 123.636,A 142.880,B 90.000,C 0.000} C_DIS
LIN {X 231.053,Y -175.256,Z 123.594,A 142.819,B 90.000,C 0.000} C_DIS
LIN {X 231.014,Y -175.306,Z 123.543,A 142.807,B 90.000,C 0.000} C_DIS
LIN {X 230.989,Y -175.340,Z 123.491,A 142.798,B 90.000,C 0.000} C_DIS
LIN {X 230.865,Y -175.503,Z 123.449,A 142.758,B 90.000,C 0.000} C_DIS
LIN {X 230.814,Y -175.570,Z 123.347,A 142.741,B 90.000,C 0.000} C_DIS
LIN {X 230.690,Y -175.733,Z 123.305,A 142.701,B 90.000,C 0.000} C_DIS
LIN {X 230.665,Y -175.767,Z 123.253,A 142.693,B 90.000,C 0.000} C_DIS
LIN {X 230.626,Y -175.817,Z 123.202,A 142.680,B 90.000,C 0.000} C_DIS
LIN {X 230.440,Y -176.061,Z 123.160,A 142.619,B 90.000,C 0.000} C_DIS
LIN {X 230.401,Y -176.111,Z 123.109,A 142.607,B 90.000,C 0.000} C_DIS
LIN {X 230.376,Y -176.145,Z 123.058,A 142.599,B 90.000,C 0.000} C_DIS
LIN {X 230.252,Y -176.307,Z 123.015,A 142.558,B 90.000,C 0.000} C_DIS
LIN {X 230.226,Y -176.341,Z 122.964,A 142.550,B 90.000,C 0.000} C_DIS
LIN {X 230.187,Y -176.391,Z 122.913,A 142.537,B 90.000,C 0.000} C_DIS
LIN {X 230.001,Y -176.634,Z 122.871,A 142.477,B 90.000,C 0.000} C_DIS
LIN {X 229.962,Y -176.685,Z 122.820,A 142.464,B 90.000,C 0.000} C_DIS
LIN {X 229.936,Y -176.718,Z 122.769,A 142.456,B 90.000,C 0.000} C_DIS
LIN {X 229.812,Y -176.880,Z 122.726,A 142.415,B 90.000,C 0.000} C_DIS
LIN {X 229.760,Y -176.948,Z 122.624,A 142.399,B 90.000,C 0.000} C_DIS
LIN {X 229.635,Y -177.109,Z 122.582,A 142.358,B 90.000,C 0.000} C_DIS
LIN {X 229.609,Y -177.143,Z 122.531,A 142.350,B 90.000,C 0.000} C_DIS
LIN {X 229.570,Y -177.193,Z 122.480,A 142.337,B 90.000,C 0.000} C_DIS
LIN {X 229.383,Y -177.436,Z 122.437,A 142.277,B 90.000,C 0.000} C_DIS
LIN {X 229.344,Y -177.486,Z 122.386,A 142.264,B 90.000,C 0.000} C_DIS
LIN {X 229.318,Y -177.520,Z 122.335,A 142.256,B 90.000,C 0.000} C_DIS
LIN {X 229.193,Y -177.681,Z 122.293,A 142.216,B 90.000,C 0.000} C_DIS
LIN {X 229.167,Y -177.715,Z 122.242,A 142.207,B 90.000,C 0.000} C_DIS
LIN {X 229.128,Y -177.765,Z 122.191,A 142.195,B 90.000,C 0.000} C_DIS
LIN {X 228.940,Y -178.007,Z 122.148,A 142.134,B 90.000,C 0.000} C_DIS
LIN {X 228.901,Y -178.057,Z 122.097,A 142.121,B 90.000,C 0.000} C_DIS
LIN {X 228.875,Y -178.090,Z 122.046,A 142.113,B 90.000,C 0.000} C_DIS
LIN {X 228.750,Y -178.252,Z 122.004,A 142.073,B 90.000,C 0.000} C_DIS
LIN {X 228.697,Y -178.318,Z 121.902,A 142.056,B 90.000,C 0.000} C_DIS
LIN {X 228.572,Y -178.479,Z 121.859,A 142.016,B 90.000,C 0.000} C_DIS
LIN {X 228.546,Y -178.513,Z 121.808,A 142.007,B 90.000,C 0.000} C_DIS
LIN {X 228.507,Y -178.563,Z 121.757,A 141.995,B 90.000,C 0.000} C_DIS
LIN {X 228.318,Y -178.804,Z 121.715,A 141.934,B 90.000,C 0.000} C_DIS
LIN {X 228.279,Y -178.854,Z 121.664,A 141.922,B 90.000,C 0.000} C_DIS
LIN {X 228.252,Y -178.888,Z 121.613,A 141.913,B 90.000,C 0.000} C_DIS
LIN {X 228.126,Y -179.048,Z 121.570,A 141.873,B 90.000,C 0.000} C_DIS
LIN {X 228.074,Y -179.115,Z 121.468,A 141.856,B 90.000,C 0.000} C_DIS
LIN {X 227.948,Y -179.276,Z 121.426,A 141.816,B 90.000,C 0.000} C_DIS
LIN {X 227.922,Y -179.309,Z 121.375,A 141.807,B 90.000,C 0.000} C_DIS
LIN {X 227.882,Y -179.359,Z 121.324,A 141.795,B 90.000,C 0.000} C_DIS
LIN {X 227.693,Y -179.600,Z 121.281,A 141.734,B 90.000,C 0.000} C_DIS
LIN {X 227.653,Y -179.650,Z 121.230,A 141.722,B 90.000,C 0.000} C_DIS
LIN {X 227.627,Y -179.683,Z 121.179,A 141.713,B 90.000,C 0.000} C_DIS
LIN {X 227.500,Y -179.843,Z 121.137,A 141.673,B 90.000,C 0.000} C_DIS
LIN {X 227.474,Y -179.877,Z 121.086,A 141.665,B 90.000,C 0.000} C_DIS
LIN {X 227.435,Y -179.926,Z 121.035,A 141.652,B 90.000,C 0.000} C_DIS
LIN {X 227.244,Y -180.167,Z 120.992,A 141.592,B 90.000,C 0.000} C_DIS
LIN {X 227.205,Y -180.216,Z 120.941,A 141.579,B 90.000,C 0.000} C_DIS
LIN {X 227.178,Y -180.250,Z 120.890,A 141.571,B 90.000,C 0.000} C_DIS
LIN {X 227.052,Y -180.410,Z 120.848,A 141.530,B 90.000,C 0.000} C_DIS
LIN {X 226.999,Y -180.476,Z 120.745,A 141.513,B 90.000,C 0.000} C_DIS
LIN {X 226.872,Y -180.636,Z 120.703,A 141.473,B 90.000,C 0.000} C_DIS
LIN {X 226.845,Y -180.669,Z 120.652,A 141.465,B 90.000,C 0.000} C_DIS
LIN {X 226.805,Y -180.719,Z 120.601,A 141.452,B 90.000,C 0.000} C_DIS
LIN {X 226.615,Y -180.958,Z 120.558,A 141.392,B 90.000,C 0.000} C_DIS
LIN {X 226.575,Y -181.008,Z 120.507,A 141.379,B 90.000,C 0.000} C_DIS
LIN {X 226.548,Y -181.041,Z 120.456,A 141.371,B 90.000,C 0.000} C_DIS
LIN {X 226.421,Y -181.201,Z 120.414,A 141.330,B 90.000,C 0.000} C_DIS
LIN {X 226.394,Y -181.234,Z 120.363,A 141.322,B 90.000,C 0.000} C_DIS
LIN {X 226.354,Y -181.283,Z 120.312,A 141.309,B 90.000,C 0.000} C_DIS
LIN {X 226.163,Y -181.522,Z 120.269,A 141.249,B 90.000,C 0.000} C_DIS
LIN {X 226.123,Y -181.572,Z 120.218,A 141.236,B 90.000,C 0.000} C_DIS
LIN {X 226.096,Y -181.605,Z 120.167,A 141.228,B 90.000,C 0.000} C_DIS
LIN {X 225.969,Y -181.764,Z 120.125,A 141.188,B 90.000,C 0.000} C_DIS
LIN {X 225.915,Y -181.830,Z 120.023,A 141.171,B 90.000,C 0.000} C_DIS
LIN {X 225.787,Y -181.989,Z 119.980,A 141.130,B 90.000,C 0.000} C_DIS
LIN {X 225.761,Y -182.022,Z 119.929,A 141.122,B 90.000,C 0.000} C_DIS
LIN {X 225.721,Y -182.072,Z 119.878,A 141.109,B 90.000,C 0.000} C_DIS
LIN {X 225.528,Y -182.310,Z 119.836,A 141.049,B 90.000,C 0.000} C_DIS
LIN {X 225.488,Y -182.360,Z 119.785,A 141.036,B 90.000,C 0.000} C_DIS
LIN {X 225.462,Y -182.393,Z 119.734,A 141.028,B 90.000,C 0.000} C_DIS
LIN {X 225.333,Y -182.551,Z 119.691,A 140.988,B 90.000,C 0.000} C_DIS
LIN {X 225.306,Y -182.584,Z 119.640,A 140.979,B 90.000,C 0.000} C_DIS
LIN {X 225.266,Y -182.634,Z 119.589,A 140.967,B 90.000,C 0.000} C_DIS
LIN {X 225.073,Y -182.872,Z 119.547,A 140.906,B 90.000,C 0.000} C_DIS
LIN {X 225.033,Y -182.921,Z 119.496,A 140.894,B 90.000,C 0.000} C_DIS
LIN {X 225.006,Y -182.954,Z 119.445,A 140.885,B 90.000,C 0.000} C_DIS
LIN {X 224.877,Y -183.112,Z 119.402,A 140.845,B 90.000,C 0.000} C_DIS
LIN {X 224.824,Y -183.178,Z 119.300,A 140.828,B 90.000,C 0.000} C_DIS
LIN {X 224.695,Y -183.336,Z 119.258,A 140.788,B 90.000,C 0.000} C_DIS
LIN {X 224.668,Y -183.369,Z 119.207,A 140.779,B 90.000,C 0.000} C_DIS
LIN {X 224.628,Y -183.419,Z 119.156,A 140.767,B 90.000,C 0.000} C_DIS
LIN {X 224.434,Y -183.656,Z 119.113,A 140.706,B 90.000,C 0.000} C_DIS
LIN {X 224.394,Y -183.705,Z 119.062,A 140.694,B 90.000,C 0.000} C_DIS
LIN {X 224.367,Y -183.738,Z 119.011,A 140.685,B 90.000,C 0.000} C_DIS
LIN {X 224.237,Y -183.896,Z 118.969,A 140.645,B 90.000,C 0.000} C_DIS
LIN {X 224.183,Y -183.961,Z 118.867,A 140.628,B 90.000,C 0.000} C_DIS
LIN {X 224.054,Y -184.119,Z 118.824,A 140.588,B 90.000,C 0.000} C_DIS
LIN {X 224.027,Y -184.152,Z 118.773,A 140.580,B 90.000,C 0.000} C_DIS
LIN {X 223.986,Y -184.201,Z 118.722,A 140.567,B 90.000,C 0.000} C_DIS
LIN {X 223.792,Y -184.438,Z 118.680,A 140.506,B 90.000,C 0.000} C_DIS
LIN {X 223.751,Y -184.487,Z 118.629,A 140.494,B 90.000,C 0.000} C_DIS
LIN {X 223.724,Y -184.519,Z 118.578,A 140.485,B 90.000,C 0.000} C_DIS
LIN {X 223.594,Y -184.677,Z 118.535,A 140.445,B 90.000,C 0.000} C_DIS
LIN {X 223.567,Y -184.710,Z 118.484,A 140.437,B 90.000,C 0.000} C_DIS
LIN {X 223.527,Y -184.759,Z 118.433,A 140.424,B 90.000,C 0.000} C_DIS
LIN {X 223.332,Y -184.995,Z 118.391,A 140.364,B 90.000,C 0.000} C_DIS
LIN {X 223.291,Y -185.044,Z 118.340,A 140.351,B 90.000,C 0.000} C_DIS
LIN {X 223.264,Y -185.076,Z 118.288,A 140.343,B 90.000,C 0.000} C_DIS
LIN {X 223.134,Y -185.233,Z 118.246,A 140.302,B 90.000,C 0.000} C_DIS
LIN {X 223.079,Y -185.299,Z 118.144,A 140.286,B 90.000,C 0.000} C_DIS
LIN {X 222.949,Y -185.456,Z 118.101,A 140.245,B 90.000,C 0.000} C_DIS
LIN {X 222.922,Y -185.488,Z 118.050,A 140.237,B 90.000,C 0.000} C_DIS
LIN {X 222.881,Y -185.537,Z 117.999,A 140.224,B 90.000,C 0.000} C_DIS
LIN {X 222.685,Y -185.773,Z 117.957,A 140.164,B 90.000,C 0.000} C_DIS
LIN {X 222.644,Y -185.822,Z 117.906,A 140.151,B 90.000,C 0.000} C_DIS
LIN {X 222.617,Y -185.854,Z 117.855,A 140.143,B 90.000,C 0.000} C_DIS
LIN {X 222.486,Y -186.011,Z 117.812,A 140.102,B 90.000,C 0.000} C_DIS
